SPLINE
SPL {X  -159.063, Y  +688.696, Z    +0.000, E1   -17.094, E3 +464723.597}
SPL {X  -159.987, Y  +672.488, Z    +0.000, E1    -5.638, E3 +464747.662}
SPL {X  -159.990, Y  +663.928, Z    +0.000, E1    +0.338, E3 +464753.456}
SPL {X  -159.990, Y  +658.009, Z    +0.000, E1    +4.774, E3 +464757.156}
SPL {X  -159.990, Y  +651.567, Z    +0.000, E1    +9.674, E3 +464762.560}
SPL {X  -159.990, Y  +638.711, Z    +0.000, E1   +17.883, E3 +464778.205}
SPL {X  -159.990, Y  +631.642, Z    +0.000, E1   +20.884, E3 +464793.764}
SPL {X  -159.990, Y  +626.048, Z    +0.000, E1   +22.026, E3 +464813.757}
SPL {X  -159.990, Y  +623.760, Z    +0.000, E1   +22.031, E3 +464825.745}
SPL {X  -159.990, Y  +621.334, Z    +0.000, E1   +22.029, E3 +464838.471}
SPL {X  -159.990, Y  +618.387, Z    +0.000, E1   +22.057, E3 +464853.861}
SPL {X  -159.990, Y  +615.830, Z    +0.000, E1   +22.023, E3 +464867.352}
SPL {X  -159.990, Y  +613.034, Z    +0.000, E1   +22.053, E3 +464881.959}
SPL {X  -159.990, Y  +609.503, Z    +0.000, E1   +22.054, E3 +464900.486}
SPL {X  -159.990, Y  +606.481, Z    +0.000, E1   +22.033, E3 +464916.360}
SPL {X  -159.990, Y  +603.419, Z    +0.000, E1   +22.064, E3 +464932.299}
SPL {X  -159.990, Y  +600.642, Z    +0.000, E1   +22.032, E3 +464946.929}
SPL {X  -159.990, Y  +598.568, Z    +0.000, E1   +22.046, E3 +464957.722}
SPL {X  -159.990, Y  +595.493, Z    +0.000, E1   +22.070, E3 +464973.805}
SPL {X  -159.990, Y  +592.865, Z    +0.000, E1   +22.036, E3 +464987.633}
SPL {X  -159.990, Y  +590.803, Z    +0.000, E1   +22.046, E3 +464998.424}
SPL {X  -159.990, Y  +587.778, Z    +0.000, E1   +22.073, E3 +465014.199}
SPL {X  -159.990, Y  +585.120, Z    +0.000, E1   +22.045, E3 +465028.143}
SPL {X  -159.990, Y  +583.118, Z    +0.000, E1   +22.052, E3 +465038.630}
SPL {X  -159.990, Y  +580.131, Z    +0.000, E1   +22.078, E3 +465054.236}
SPL {X  -159.990, Y  +576.888, Z    +0.000, E1   +22.061, E3 +465071.266}
SPL {X  -159.990, Y  +574.280, Z    +0.000, E1   +22.051, E3 +465084.940}
SPL {X  -159.990, Y  +572.375, Z    +0.000, E1   +22.037, E3 +465094.978}
SPL {X  -159.990, Y  +569.881, Z    +0.000, E1   +22.067, E3 +465107.973}
SPL {X  -159.990, Y  +567.211, Z    +0.000, E1   +22.046, E3 +465122.000}
SPL {X  -159.990, Y  +565.039, Z    +0.000, E1   +22.047, E3 +465133.377}
SPL {X  -159.990, Y  +562.755, Z    +0.000, E1   +22.047, E3 +465145.363}
SPL {X  -159.990, Y  +560.652, Z    +0.000, E1   +22.038, E3 +465156.408}
SPL {X  -159.990, Y  +558.852, Z    +0.000, E1   +22.046, E3 +465165.779}
SPL {X  -159.990, Y  +556.672, Z    +0.000, E1   +22.055, E3 +465177.169}
SPL {X  -159.990, Y  +553.726, Z    +0.000, E1   +22.080, E3 +465192.531}
SPL {X  -159.990, Y  +550.886, Z    +0.000, E1   +22.056, E3 +465207.470}
SPL {X  -159.990, Y  +548.814, Z    +0.000, E1   +22.049, E3 +465218.316}
SPL {X  -159.990, Y  +546.122, Z    +0.000, E1   +22.088, E3 +465232.330}
SPL {X  -159.990, Y  +542.390, Z    +0.000, E1   +22.086, E3 +465251.912}
SPL {X  -159.990, Y  +539.341, Z    +0.000, E1   +22.056, E3 +465267.933}
SPL {X  -159.990, Y  +536.984, Z    +0.000, E1   +22.057, E3 +465280.264}
SPL {X  -159.990, Y  +534.045, Z    +0.000, E1   +22.087, E3 +465295.589}
SPL {X  -159.990, Y  +530.476, Z    +0.000, E1   +22.084, E3 +465314.282}
SPL {X  -159.990, Y  +527.412, Z    +0.000, E1   +22.067, E3 +465330.346}
SPL {X  -159.990, Y  +525.349, Z    +0.000, E1   +22.050, E3 +465341.187}
SPL {X  -159.990, Y  +523.717, Z    +0.000, E1   +22.050, E3 +465349.752}
SPL {X  -159.990, Y  +521.599, Z    +0.000, E1   +22.060, E3 +465360.820}
SPL {X  -159.990, Y  +519.209, Z    +0.000, E1   +22.063, E3 +465373.295}
SPL {X  -159.990, Y  +517.330, Z    +0.000, E1   +22.053, E3 +465383.151}
SPL {X  -159.990, Y  +514.729, Z    +0.000, E1   +22.089, E3 +465396.709}
SPL {X  -159.990, Y  +511.670, Z    +0.000, E1   +22.064, E3 +465412.796}
SPL {X  -159.990, Y  +506.947, Z    +0.000, E1   +23.726, E3 +465422.825}
SPL {X  -159.990, Y  +496.921, Z    +0.000, E1   +28.340, E3 +465431.573}
SPL {X  -159.990, Y  +495.822, Z    +0.000, E1   +27.449, E3 +465442.321}
SPL {X  -159.990, Y  +494.952, Z    +0.000, E1   +26.628, E3 +465451.905}
SPL {X  -159.990, Y  +493.896, Z    +0.000, E1   +25.736, E3 +465463.234}
SPL {X  -159.990, Y  +491.647, Z    +0.000, E1   +25.401, E3 +465475.770}
SPL {X  -159.990, Y  +488.807, Z    +0.000, E1   +25.397, E3 +465488.468}
SPL {X  -159.990, Y  +486.070, Z    +0.000, E1   +25.399, E3 +465500.699}
SPL {X  -159.990, Y  +482.821, Z    +0.000, E1   +25.411, E3 +465515.201}
SPL {X  -159.990, Y  +480.183, Z    +0.000, E1   +25.384, E3 +465527.041}
SPL {X  -159.990, Y  +477.508, Z    +0.000, E1   +25.410, E3 +465538.950}
SPL {X  -159.990, Y  +473.634, Z    +0.000, E1   +25.426, E3 +465556.239}
SPL {X  -159.990, Y  +470.047, Z    +0.000, E1   +25.402, E3 +465572.320}
SPL {X  -159.990, Y  +467.082, Z    +0.000, E1   +25.399, E3 +465585.567}
SPL {X  -159.990, Y  +464.063, Z    +0.000, E1   +25.405, E3 +465599.062}
SPL {X  -159.990, Y  +460.712, Z    +0.000, E1   +25.411, E3 +465614.022}
SPL {X  -159.990, Y  +457.497, Z    +0.000, E1   +25.403, E3 +465628.394}
SPL {X  -159.990, Y  +455.126, Z    +0.000, E1   +25.389, E3 +465639.002}
SPL {X  -159.990, Y  +453.438, Z    +0.000, E1   +25.385, E3 +465646.562}
SPL {X  -159.990, Y  +450.823, Z    +0.000, E1   +25.417, E3 +465658.182}
SPL {X  -159.990, Y  +446.894, Z    +0.000, E1   +25.428, E3 +465675.739}
SPL {X  -159.990, Y  +443.345, Z    +0.000, E1   +25.390, E3 +465691.746}
SPL {X  -159.990, Y  +441.077, Z    +0.000, E1   +25.369, E3 +465701.945}
SPL {X  -159.990, Y  +438.608, Z    +0.000, E1   +25.392, E3 +465712.941}
SPL {X  -159.990, Y  +434.852, Z    +0.000, E1   +25.415, E3 +465729.696}
SPL {X  -159.990, Y  +430.645, Z    +0.000, E1   +25.414, E3 +465748.515}
SPL {X  -159.990, Y  +426.865, Z    +0.000, E1   +25.398, E3 +465765.445}
SPL {X  -159.990, Y  +424.251, Z    +0.000, E1   +25.375, E3 +465777.182}
SPL {X  -159.990, Y  +421.010, Z    +0.000, E1   +25.418, E3 +465791.597}
SPL {X  -159.990, Y  +417.514, Z    +0.000, E1   +25.386, E3 +465807.290}
SPL {X  -159.990, Y  +414.805, Z    +0.000, E1   +25.385, E3 +465819.410}
SPL {X  -159.990, Y  +411.959, Z    +0.000, E1   +25.386, E3 +465832.137}
SPL {X  -159.990, Y  +408.981, Z    +0.000, E1   +25.392, E3 +465845.440}
SPL {X  -159.990, Y  +406.574, Z    +0.000, E1   +25.375, E3 +465856.214}
SPL {X  -159.990, Y  +403.513, Z    +0.000, E1   +25.420, E3 +465869.813}
SPL {X  -159.990, Y  +399.257, Z    +0.000, E1   +25.420, E3 +465888.854}
SPL {X  -159.990, Y  +395.992, Z    +0.000, E1   +25.380, E3 +465903.544}
SPL {X  -159.990, Y  +393.569, Z    +0.000, E1   +25.379, E3 +465914.387}
SPL {X  -159.990, Y  +390.564, Z    +0.000, E1   +25.393, E3 +465927.831}
SPL {X  -159.990, Y  +387.503, Z    +0.000, E1   +25.378, E3 +465941.546}
SPL {X  -159.990, Y  +384.900, Z    +0.000, E1   +25.383, E3 +465953.156}
SPL {X  -159.990, Y  +382.110, Z    +0.000, E1   +25.393, E3 +465965.602}
SPL {X  -159.961, Y  +379.439, Z    +0.000, E1   +25.380, E3 +465977.582}
SPL {X  -159.894, Y  +376.959, Z    +0.000, E1   +25.370, E3 +465988.759}
SPL {X  -159.784, Y  +374.382, Z    +0.000, E1   +25.356, E3 +466000.399}
SPL {X  -159.621, Y  +371.640, Z    +0.000, E1   +25.335, E3 +466012.839}
SPL {X  -159.406, Y  +368.844, Z    +0.000, E1   +25.307, E3 +466025.552}
SPL {X  -159.144, Y  +366.072, Z    +0.000, E1   +25.281, E3 +466038.160}
SPL {X  -158.822, Y  +363.200, Z    +0.000, E1   +25.236, E3 +466051.333}
SPL {X  -158.491, Y  +360.654, Z    +0.000, E1   +25.188, E3 +466063.073}
SPL {X  -158.127, Y  +358.155, Z    +0.000, E1   +25.126, E3 +466074.692}
SPL {X  -158.095, Y  +357.947, Z    +0.000, E1   +21.741, E3 +466106.265}
ENDSPLINE

SPLINE
SPL {X  -158.454, Y  +360.384, Z    +0.000, E1   +19.366, E3 +466118.416}
SPL {X  -159.737, Y  +373.507, Z    +0.000, E1   +10.311, E3 +466140.451}
SPL {X  -159.990, Y  +382.574, Z    +0.000, E1    +4.463, E3 +466147.139}
SPL {X  -159.990, Y  +387.496, Z    +0.000, E1    +1.004, E3 +466149.884}
SPL {X  -159.990, Y  +395.121, Z    +0.000, E1    -4.514, E3 +466154.196}
SPL {X  -159.990, Y  +407.941, Z    +0.000, E1   -14.126, E3 +466166.270}
SPL {X  -159.990, Y  +418.671, Z    +0.000, E1   -19.855, E3 +466185.687}
SPL {X  -159.990, Y  +429.878, Z    +0.000, E1   -23.330, E3 +466215.742}
SPL {X  -159.990, Y  +432.766, Z    +0.000, E1   -23.321, E3 +466229.964}
SPL {X  -159.990, Y  +434.794, Z    +0.000, E1   -23.304, E3 +466239.996}
SPL {X  -159.990, Y  +437.007, Z    +0.000, E1   -23.323, E3 +466250.848}
SPL {X  -159.990, Y  +439.778, Z    +0.000, E1   -23.323, E3 +466264.480}
SPL {X  -159.990, Y  +442.010, Z    +0.000, E1   -23.308, E3 +466275.501}
SPL {X  -159.990, Y  +443.729, Z    +0.000, E1   -23.310, E3 +466283.958}
SPL {X  -159.990, Y  +446.037, Z    +0.000, E1   -23.324, E3 +466295.295}
SPL {X  -159.990, Y  +449.434, Z    +0.000, E1   -23.356, E3 +466311.916}
SPL {X  -159.990, Y  +453.256, Z    +0.000, E1   -23.349, E3 +466330.751}
SPL {X  -159.990, Y  +455.953, Z    +0.000, E1   -23.320, E3 +466344.065}
SPL {X  -159.990, Y  +458.265, Z    +0.000, E1   -23.328, E3 +466355.420}
SPL {X  -159.990, Y  +460.492, Z    +0.000, E1   -23.317, E3 +466366.419}
SPL {X  -159.990, Y  +462.929, Z    +0.000, E1   -23.331, E3 +466378.375}
SPL {X  -159.990, Y  +466.197, Z    +0.000, E1   -23.351, E3 +466394.412}
SPL {X  -159.990, Y  +468.951, Z    +0.000, E1   -23.319, E3 +466408.029}
SPL {X  -159.990, Y  +470.991, Z    +0.000, E1   -23.322, E3 +466418.059}
SPL {X  -159.990, Y  +474.027, Z    +0.000, E1   -23.352, E3 +466432.963}
SPL {X  -159.990, Y  +476.830, Z    +0.000, E1   -23.323, E3 +466446.830}
SPL {X  -159.990, Y  +479.553, Z    +0.000, E1   -23.328, E3 +466460.233}
SPL {X  -159.990, Y  +482.950, Z    +0.000, E1   -23.350, E3 +466476.905}
SPL {X  -159.990, Y  +486.109, Z    +0.000, E1   -23.322, E3 +466492.520}
SPL {X  -159.990, Y  +488.481, Z    +0.000, E1   -23.319, E3 +466504.200}
SPL {X  -159.990, Y  +491.454, Z    +0.000, E1   -23.343, E3 +466518.780}
SPL {X  -159.990, Y  +494.937, Z    +0.000, E1   -23.343, E3 +466535.924}
SPL {X  -159.990, Y  +497.668, Z    +0.000, E1   -23.317, E3 +466549.418}
SPL {X  -159.990, Y  +499.995, Z    +0.000, E1   -23.324, E3 +466560.855}
SPL {X  -159.990, Y  +502.456, Z    +0.000, E1   -23.324, E3 +466572.970}
SPL {X  -159.990, Y  +504.508, Z    +0.000, E1   -23.311, E3 +466583.104}
SPL {X  -159.990, Y  +506.420, Z    +0.000, E1   -23.317, E3 +466592.497}
SPL {X  -159.990, Y  +508.862, Z    +0.000, E1   -23.328, E3 +466604.490}
SPL {X  -159.990, Y  +511.771, Z    +0.000, E1   -23.331, E3 +466618.811}
SPL {X  -159.990, Y  +514.016, Z    +0.000, E1   -23.308, E3 +466629.915}
SPL {X  -159.990, Y  +516.860, Z    +0.000, E1   -23.355, E3 +466643.801}
SPL {X  -159.990, Y  +520.719, Z    +0.000, E1   -23.363, E3 +466662.712}
SPL {X  -159.990, Y  +523.968, Z    +0.000, E1   -23.332, E3 +466678.797}
SPL {X  -159.990, Y  +526.466, Z    +0.000, E1   -23.320, E3 +466691.140}
SPL {X  -159.990, Y  +528.815, Z    +0.000, E1   -23.322, E3 +466702.699}
SPL {X  -159.990, Y  +531.246, Z    +0.000, E1   -23.325, E3 +466714.638}
SPL {X  -159.990, Y  +534.143, Z    +0.000, E1   -23.341, E3 +466728.873}
SPL {X  -159.990, Y  +537.024, Z    +0.000, E1   -23.321, E3 +466743.116}
SPL {X  -159.990, Y  +539.129, Z    +0.000, E1   -23.310, E3 +466753.499}
SPL {X  -159.990, Y  +541.882, Z    +0.000, E1   -23.346, E3 +466766.980}
SPL {X  -159.990, Y  +544.941, Z    +0.000, E1   -23.325, E3 +466782.063}
SPL {X  -159.990, Y  +547.390, Z    +0.000, E1   -23.325, E3 +466794.116}
SPL {X  -159.990, Y  +550.708, Z    +0.000, E1   -23.357, E3 +466810.383}
SPL {X  -159.990, Y  +553.642, Z    +0.000, E1   -23.319, E3 +466824.890}
SPL {X  -159.990, Y  +555.637, Z    +0.000, E1   -23.323, E3 +466834.704}
SPL {X  -159.990, Y  +558.758, Z    +0.000, E1   -23.351, E3 +466850.014}
SPL {X  -159.990, Y  +561.830, Z    +0.000, E1   -23.325, E3 +466865.187}
SPL {X  -159.990, Y  +564.273, Z    +0.000, E1   -23.325, E3 +466877.212}
SPL {X  -159.990, Y  +567.351, Z    +0.000, E1   -23.348, E3 +466892.307}
SPL {X  -159.990, Y  +570.560, Z    +0.000, E1   -23.333, E3 +466908.137}
SPL {X  -159.990, Y  +572.975, Z    +0.000, E1   -23.316, E3 +466920.056}
SPL {X  -159.990, Y  +575.097, Z    +0.000, E1   -23.325, E3 +466930.483}
SPL {X  -159.990, Y  +578.356, Z    +0.000, E1   -23.358, E3 +466946.455}
SPL {X  -159.990, Y  +582.292, Z    +0.000, E1   -23.360, E3 +466965.771}
SPL {X  -159.990, Y  +585.165, Z    +0.000, E1   -23.322, E3 +466980.014}
SPL {X  -159.990, Y  +587.388, Z    +0.000, E1   -23.328, E3 +466990.927}
SPL {X  -159.990, Y  +589.763, Z    +0.000, E1   -23.328, E3 +467002.614}
SPL {X  -159.990, Y  +592.397, Z    +0.000, E1   -23.344, E3 +467015.495}
SPL {X  -159.990, Y  +595.589, Z    +0.000, E1   -23.356, E3 +467031.167}
SPL {X  -159.990, Y  +598.571, Z    +0.000, E1   -23.347, E3 +467045.811}
SPL {X  -159.990, Y  +600.935, Z    +0.000, E1   -23.343, E3 +467057.404}
SPL {X  -159.990, Y  +603.047, Z    +0.000, E1   -23.344, E3 +467067.790}
SPL {X  -159.990, Y  +605.187, Z    +0.000, E1   -23.344, E3 +467078.311}
SPL {X  -159.990, Y  +607.319, Z    +0.000, E1   -23.353, E3 +467088.774}
SPL {X  -159.990, Y  +609.514, Z    +0.000, E1   -23.337, E3 +467099.603}
SPL {X  -159.990, Y  +611.376, Z    +0.000, E1   -23.336, E3 +467108.790}
SPL {X  -159.990, Y  +613.591, Z    +0.000, E1   -23.342, E3 +467119.667}
SPL {X  -159.990, Y  +615.604, Z    +0.000, E1   -23.330, E3 +467129.605}
SPL {X  -159.990, Y  +617.623, Z    +0.000, E1   -23.337, E3 +467139.535}
SPL {X  -159.990, Y  +620.788, Z    +0.000, E1   -23.368, E3 +467155.041}
SPL {X  -159.990, Y  +623.764, Z    +0.000, E1   -23.335, E3 +467169.733}
SPL {X  -159.990, Y  +625.941, Z    +0.000, E1   -23.337, E3 +467180.424}
SPL {X  -159.990, Y  +628.611, Z    +0.000, E1   -23.357, E3 +467193.503}
SPL {X  -159.990, Y  +631.169, Z    +0.000, E1   -23.338, E3 +467206.107}
SPL {X  -159.990, Y  +633.318, Z    +0.000, E1   -23.339, E3 +467216.697}
SPL {X  -159.990, Y  +635.650, Z    +0.000, E1   -23.339, E3 +467228.167}
SPL {X  -159.990, Y  +637.839, Z    +0.000, E1   -23.335, E3 +467238.978}
SPL {X  -159.990, Y  +640.072, Z    +0.000, E1   -23.325, E3 +467250.010}
SPL {X  -159.990, Y  +642.230, Z    +0.000, E1   -23.323, E3 +467260.691}
SPL {X  -159.990, Y  +645.287, Z    +0.000, E1   -23.340, E3 +467275.717}
SPL {X  -159.990, Y  +647.803, Z    +0.000, E1   -23.310, E3 +467288.194}
SPL {X  -159.990, Y  +650.790, Z    +0.000, E1   -23.346, E3 +467302.802}
SPL {X  -159.990, Y  +654.543, Z    +0.000, E1   -23.348, E3 +467321.255}
SPL {X  -159.990, Y  +658.319, Z    +0.000, E1   -23.349, E3 +467339.844}
SPL {X  -159.990, Y  +661.392, Z    +0.000, E1   -23.318, E3 +467355.047}
SPL {X  -159.990, Y  +663.662, Z    +0.000, E1   -23.322, E3 +467366.172}
SPL {X  -159.990, Y  +665.964, Z    +0.000, E1   -23.328, E3 +467377.462}
SPL {X  -159.990, Y  +667.870, Z    +0.000, E1   -23.320, E3 +467386.869}
SPL {X  -159.990, Y  +669.861, Z    +0.000, E1   -23.321, E3 +467396.670}
SPL {X  -159.990, Y  +671.893, Z    +0.000, E1   -23.319, E3 +467406.678}
SPL {X  -159.974, Y  +673.789, Z    +0.000, E1   -23.323, E3 +467415.994}
SPL {X  -159.924, Y  +676.110, Z    +0.000, E1   -23.320, E3 +467427.478}
SPL {X  -159.801, Y  +679.265, Z    +0.000, E1   -23.327, E3 +467443.097}
SPL {X  -159.626, Y  +682.287, Z    +0.000, E1   -23.280, E3 +467458.195}
SPL {X  -159.462, Y  +684.486, Z    +0.000, E1   -23.258, E3 +467469.195}
SPL {X  -159.246, Y  +686.911, Z    +0.000, E1   -23.230, E3 +467481.356}
SPL {X  -159.019, Y  +689.098, Z    +0.000, E1   -23.200, E3 +467492.358}
SPL {X  -158.660, Y  +692.086, Z    +0.000, E1   -23.176, E3 +467507.402}
ENDSPLINE

SPLINE
SPL {X  -159.063, Y  +688.696, Z    +0.000, E1   -17.094, E3 +467549.684}
SPL {X  -159.967, Y  +674.206, Z    +0.000, E1    -6.731, E3 +467572.496}
SPL {X  -159.990, Y  +665.270, Z    +0.000, E1    -0.699, E3 +467578.666}
SPL {X  -159.990, Y  +658.009, Z    +0.000, E1    +4.774, E3 +467583.243}
SPL {X  -159.990, Y  +651.567, Z    +0.000, E1    +9.674, E3 +467588.647}
SPL {X  -159.990, Y  +638.711, Z    +0.000, E1   +17.883, E3 +467604.292}
SPL {X  -159.990, Y  +631.642, Z    +0.000, E1   +20.884, E3 +467619.851}
SPL {X  -159.990, Y  +626.048, Z    +0.000, E1   +22.026, E3 +467639.844}
SPL {X  -159.990, Y  +623.760, Z    +0.000, E1   +22.031, E3 +467651.832}
SPL {X  -159.990, Y  +621.334, Z    +0.000, E1   +22.029, E3 +467664.558}
SPL {X  -159.990, Y  +618.387, Z    +0.000, E1   +22.057, E3 +467679.948}
SPL {X  -159.990, Y  +614.928, Z    +0.000, E1   +22.055, E3 +467698.101}
SPL {X  -159.990, Y  +611.459, Z    +0.000, E1   +22.053, E3 +467716.304}
SPL {X  -159.990, Y  +608.810, Z    +0.000, E1   +22.023, E3 +467730.271}
SPL {X  -159.990, Y  +606.481, Z    +0.000, E1   +22.033, E3 +467742.447}
SPL {X  -159.990, Y  +603.419, Z    +0.000, E1   +22.064, E3 +467758.386}
SPL {X  -159.990, Y  +600.642, Z    +0.000, E1   +22.032, E3 +467773.016}
SPL {X  -159.990, Y  +598.568, Z    +0.000, E1   +22.046, E3 +467783.809}
SPL {X  -159.990, Y  +596.440, Z    +0.000, E1   +22.036, E3 +467794.990}
SPL {X  -159.990, Y  +593.768, Z    +0.000, E1   +22.071, E3 +467808.923}
SPL {X  -159.990, Y  +590.803, Z    +0.000, E1   +22.046, E3 +467824.511}
SPL {X  -159.990, Y  +587.778, Z    +0.000, E1   +22.073, E3 +467840.286}
SPL {X  -159.990, Y  +585.120, Z    +0.000, E1   +22.045, E3 +467854.230}
SPL {X  -159.990, Y  +583.118, Z    +0.000, E1   +22.052, E3 +467864.717}
SPL {X  -159.990, Y  +580.131, Z    +0.000, E1   +22.078, E3 +467880.323}
SPL {X  -159.990, Y  +576.888, Z    +0.000, E1   +22.061, E3 +467897.353}
SPL {X  -159.990, Y  +574.280, Z    +0.000, E1   +22.051, E3 +467911.027}
SPL {X  -159.990, Y  +572.375, Z    +0.000, E1   +22.037, E3 +467921.065}
SPL {X  -159.990, Y  +569.881, Z    +0.000, E1   +22.067, E3 +467934.059}
SPL {X  -159.990, Y  +567.211, Z    +0.000, E1   +22.046, E3 +467948.087}
SPL {X  -159.990, Y  +565.039, Z    +0.000, E1   +22.047, E3 +467959.464}
SPL {X  -159.990, Y  +562.755, Z    +0.000, E1   +22.047, E3 +467971.449}
SPL {X  -159.990, Y  +559.661, Z    +0.000, E1   +22.078, E3 +467987.581}
SPL {X  -159.990, Y  +555.965, Z    +0.000, E1   +22.085, E3 +468006.890}
SPL {X  -159.990, Y  +553.115, Z    +0.000, E1   +22.054, E3 +468021.876}
SPL {X  -159.990, Y  +550.886, Z    +0.000, E1   +22.056, E3 +468033.557}
SPL {X  -159.990, Y  +547.986, Z    +0.000, E1   +22.078, E3 +468048.677}
SPL {X  -159.990, Y  +545.350, Z    +0.000, E1   +22.053, E3 +468062.538}
SPL {X  -159.990, Y  +543.405, Z    +0.000, E1   +22.048, E3 +468072.751}
SPL {X  -159.990, Y  +541.673, Z    +0.000, E1   +22.053, E3 +468081.815}
SPL {X  -159.990, Y  +539.341, Z    +0.000, E1   +22.056, E3 +468094.020}
SPL {X  -159.990, Y  +536.301, Z    +0.000, E1   +22.084, E3 +468109.875}
SPL {X  -159.990, Y  +533.389, Z    +0.000, E1   +22.057, E3 +468125.182}
SPL {X  -159.990, Y  +531.347, Z    +0.000, E1   +22.052, E3 +468135.883}
SPL {X  -159.990, Y  +529.626, Z    +0.000, E1   +22.051, E3 +468144.880}
SPL {X  -159.990, Y  +527.412, Z    +0.000, E1   +22.067, E3 +468156.432}
SPL {X  -159.990, Y  +524.425, Z    +0.000, E1   +22.078, E3 +468172.065}
SPL {X  -159.990, Y  +521.599, Z    +0.000, E1   +22.060, E3 +468186.907}
SPL {X  -159.990, Y  +519.209, Z    +0.000, E1   +22.063, E3 +468199.382}
SPL {X  -159.990, Y  +516.651, Z    +0.000, E1   +22.071, E3 +468212.761}
SPL {X  -159.990, Y  +514.122, Z    +0.000, E1   +22.061, E3 +468226.033}
SPL {X  -159.990, Y  +511.670, Z    +0.000, E1   +22.064, E3 +468238.883}
SPL {X  -159.990, Y  +506.947, Z    +0.000, E1   +23.726, E3 +468248.912}
SPL {X  -159.990, Y  +496.921, Z    +0.000, E1   +28.340, E3 +468257.660}
SPL {X  -159.990, Y  +495.822, Z    +0.000, E1   +27.449, E3 +468268.408}
SPL {X  -159.990, Y  +494.952, Z    +0.000, E1   +26.628, E3 +468277.992}
SPL {X  -159.990, Y  +493.896, Z    +0.000, E1   +25.736, E3 +468289.321}
SPL {X  -159.990, Y  +491.647, Z    +0.000, E1   +25.401, E3 +468301.857}
SPL {X  -159.990, Y  +488.807, Z    +0.000, E1   +25.397, E3 +468314.555}
SPL {X  -159.990, Y  +486.070, Z    +0.000, E1   +25.399, E3 +468326.786}
SPL {X  -159.990, Y  +483.747, Z    +0.000, E1   +25.384, E3 +468337.199}
SPL {X  -159.990, Y  +481.980, Z    +0.000, E1   +25.384, E3 +468345.097}
SPL {X  -159.990, Y  +479.252, Z    +0.000, E1   +25.412, E3 +468357.238}
SPL {X  -159.990, Y  +475.940, Z    +0.000, E1   +25.403, E3 +468372.059}
SPL {X  -159.990, Y  +473.026, Z    +0.000, E1   +25.399, E3 +468385.088}
SPL {X  -159.990, Y  +470.047, Z    +0.000, E1   +25.402, E3 +468398.407}
SPL {X  -159.990, Y  +466.213, Z    +0.000, E1   +25.433, E3 +468415.486}
SPL {X  -159.990, Y  +462.520, Z    +0.000, E1   +25.400, E3 +468432.055}
SPL {X  -159.990, Y  +460.081, Z    +0.000, E1   +25.390, E3 +468442.956}
SPL {X  -159.990, Y  +457.497, Z    +0.000, E1   +25.403, E3 +468454.481}
SPL {X  -159.990, Y  +455.126, Z    +0.000, E1   +25.389, E3 +468465.089}
SPL {X  -159.990, Y  +452.123, Z    +0.000, E1   +25.426, E3 +468478.447}
SPL {X  -159.990, Y  +448.503, Z    +0.000, E1   +25.410, E3 +468494.648}
SPL {X  -159.990, Y  +445.882, Z    +0.000, E1   +25.385, E3 +468506.451}
SPL {X  -159.990, Y  +443.345, Z    +0.000, E1   +25.390, E3 +468517.833}
SPL {X  -159.990, Y  +441.077, Z    +0.000, E1   +25.369, E3 +468528.032}
SPL {X  -159.990, Y  +438.608, Z    +0.000, E1   +25.392, E3 +468539.028}
SPL {X  -159.990, Y  +434.852, Z    +0.000, E1   +25.415, E3 +468555.783}
SPL {X  -159.990, Y  +430.645, Z    +0.000, E1   +25.414, E3 +468574.602}
SPL {X  -159.990, Y  +426.865, Z    +0.000, E1   +25.398, E3 +468591.532}
SPL {X  -159.990, Y  +424.251, Z    +0.000, E1   +25.375, E3 +468603.269}
SPL {X  -159.990, Y  +421.010, Z    +0.000, E1   +25.418, E3 +468617.684}
SPL {X  -159.990, Y  +417.514, Z    +0.000, E1   +25.386, E3 +468633.377}
SPL {X  -159.990, Y  +414.805, Z    +0.000, E1   +25.385, E3 +468645.497}
SPL {X  -159.990, Y  +411.282, Z    +0.000, E1   +25.413, E3 +468661.198}
SPL {X  -159.990, Y  +408.351, Z    +0.000, E1   +25.372, E3 +468674.385}
SPL {X  -159.990, Y  +405.773, Z    +0.000, E1   +25.398, E3 +468685.837}
SPL {X  -159.990, Y  +402.805, Z    +0.000, E1   +25.389, E3 +468699.123}
SPL {X  -159.990, Y  +400.083, Z    +0.000, E1   +25.388, E3 +468711.300}
SPL {X  -159.990, Y  +396.740, Z    +0.000, E1   +25.410, E3 +468726.224}
SPL {X  -159.990, Y  +392.622, Z    +0.000, E1   +25.413, E3 +468744.652}
SPL {X  -159.990, Y  +388.328, Z    +0.000, E1   +25.413, E3 +468763.881}
SPL {X  -159.990, Y  +384.900, Z    +0.000, E1   +25.383, E3 +468779.243}
SPL {X  -159.990, Y  +382.110, Z    +0.000, E1   +25.393, E3 +468791.689}
SPL {X  -159.961, Y  +379.439, Z    +0.000, E1   +25.380, E3 +468803.669}
SPL {X  -159.894, Y  +376.959, Z    +0.000, E1   +25.370, E3 +468814.846}
SPL {X  -159.784, Y  +374.382, Z    +0.000, E1   +25.356, E3 +468826.486}
SPL {X  -159.621, Y  +371.640, Z    +0.000, E1   +25.335, E3 +468838.926}
SPL {X  -159.406, Y  +368.844, Z    +0.000, E1   +25.307, E3 +468851.639}
SPL {X  -159.144, Y  +366.072, Z    +0.000, E1   +25.281, E3 +468864.247}
SPL {X  -158.822, Y  +363.200, Z    +0.000, E1   +25.236, E3 +468877.420}
SPL {X  -158.491, Y  +360.654, Z    +0.000, E1   +25.188, E3 +468889.160}
SPL {X  -158.127, Y  +358.155, Z    +0.000, E1   +25.126, E3 +468900.779}
SPL {X  -158.095, Y  +357.947, Z    +0.000, E1   +21.741, E3 +468932.352}
ENDSPLINE

SPLINE
SPL {X  -158.454, Y  +360.384, Z    +0.000, E1   +19.366, E3 +468944.503}
SPL {X  -159.737, Y  +373.507, Z    +0.000, E1   +10.311, E3 +468966.538}
SPL {X  -159.990, Y  +382.574, Z    +0.000, E1    +4.463, E3 +468973.226}
SPL {X  -159.990, Y  +389.909, Z    +0.000, E1    -0.662, E3 +468977.240}
SPL {X  -159.990, Y  +396.289, Z    +0.000, E1    -5.500, E3 +468981.020}
SPL {X  -159.990, Y  +407.941, Z    +0.000, E1   -14.126, E3 +468992.357}
SPL {X  -159.990, Y  +418.671, Z    +0.000, E1   -19.855, E3 +469011.774}
SPL {X  -159.990, Y  +429.878, Z    +0.000, E1   -23.330, E3 +469041.829}
SPL {X  -159.990, Y  +432.103, Z    +0.000, E1   -23.301, E3 +469052.847}
SPL {X  -159.990, Y  +434.188, Z    +0.000, E1   -23.325, E3 +469063.044}
SPL {X  -159.990, Y  +437.007, Z    +0.000, E1   -23.323, E3 +469076.935}
SPL {X  -159.990, Y  +439.778, Z    +0.000, E1   -23.323, E3 +469090.567}
SPL {X  -159.990, Y  +442.945, Z    +0.000, E1   -23.339, E3 +469106.131}
SPL {X  -159.990, Y  +446.037, Z    +0.000, E1   -23.324, E3 +469121.382}
SPL {X  -159.990, Y  +448.797, Z    +0.000, E1   -23.331, E3 +469134.912}
SPL {X  -159.990, Y  +451.747, Z    +0.000, E1   -23.333, E3 +469149.460}
SPL {X  -159.990, Y  +454.210, Z    +0.000, E1   -23.316, E3 +469161.591}
SPL {X  -159.990, Y  +455.953, Z    +0.000, E1   -23.320, E3 +469170.152}
SPL {X  -159.990, Y  +458.265, Z    +0.000, E1   -23.328, E3 +469181.507}
SPL {X  -159.990, Y  +461.258, Z    +0.000, E1   -23.344, E3 +469196.223}
SPL {X  -159.990, Y  +464.382, Z    +0.000, E1   -23.332, E3 +469211.604}
SPL {X  -159.990, Y  +466.881, Z    +0.000, E1   -23.322, E3 +469223.924}
SPL {X  -159.990, Y  +468.951, Z    +0.000, E1   -23.319, E3 +469234.116}
SPL {X  -159.990, Y  +470.991, Z    +0.000, E1   -23.322, E3 +469244.146}
SPL {X  -159.990, Y  +474.027, Z    +0.000, E1   -23.352, E3 +469259.050}
SPL {X  -159.990, Y  +477.600, Z    +0.000, E1   -23.351, E3 +469276.653}
SPL {X  -159.990, Y  +481.169, Z    +0.000, E1   -23.337, E3 +469294.250}
SPL {X  -159.990, Y  +483.782, Z    +0.000, E1   -23.316, E3 +469307.155}
SPL {X  -159.990, Y  +486.109, Z    +0.000, E1   -23.322, E3 +469318.607}
SPL {X  -159.990, Y  +489.247, Z    +0.000, E1   -23.348, E3 +469333.995}
SPL {X  -159.990, Y  +493.031, Z    +0.000, E1   -23.350, E3 +469352.619}
SPL {X  -159.990, Y  +496.869, Z    +0.000, E1   -23.349, E3 +469371.509}
SPL {X  -159.990, Y  +499.995, Z    +0.000, E1   -23.324, E3 +469386.942}
SPL {X  -159.990, Y  +502.456, Z    +0.000, E1   -23.324, E3 +469399.057}
SPL {X  -159.990, Y  +505.646, Z    +0.000, E1   -23.350, E3 +469414.712}
SPL {X  -159.990, Y  +508.862, Z    +0.000, E1   -23.328, E3 +469430.577}
SPL {X  -159.990, Y  +510.971, Z    +0.000, E1   -23.308, E3 +469441.004}
SPL {X  -159.990, Y  +512.484, Z    +0.000, E1   -23.309, E3 +469448.454}
SPL {X  -159.990, Y  +514.757, Z    +0.000, E1   -23.329, E3 +469459.606}
SPL {X  -159.990, Y  +517.536, Z    +0.000, E1   -23.326, E3 +469473.273}
SPL {X  -159.990, Y  +519.961, Z    +0.000, E1   -23.334, E3 +469485.125}
SPL {X  -159.990, Y  +521.849, Z    +0.000, E1   -23.320, E3 +469494.448}
SPL {X  -159.990, Y  +523.968, Z    +0.000, E1   -23.332, E3 +469504.883}
SPL {X  -159.990, Y  +526.466, Z    +0.000, E1   -23.320, E3 +469517.227}
SPL {X  -159.990, Y  +528.815, Z    +0.000, E1   -23.322, E3 +469528.786}
SPL {X  -159.990, Y  +531.246, Z    +0.000, E1   -23.325, E3 +469540.725}
SPL {X  -159.990, Y  +533.354, Z    +0.000, E1   -23.318, E3 +469551.110}
SPL {X  -159.990, Y  +534.931, Z    +0.000, E1   -23.312, E3 +469558.905}
SPL {X  -159.990, Y  +537.024, Z    +0.000, E1   -23.321, E3 +469569.203}
SPL {X  -159.990, Y  +539.129, Z    +0.000, E1   -23.310, E3 +469579.586}
SPL {X  -159.990, Y  +541.183, Z    +0.000, E1   -23.319, E3 +469589.683}
SPL {X  -159.990, Y  +544.314, Z    +0.000, E1   -23.352, E3 +469605.011}
SPL {X  -159.990, Y  +548.126, Z    +0.000, E1   -23.354, E3 +469623.767}
SPL {X  -159.990, Y  +551.344, Z    +0.000, E1   -23.327, E3 +469639.659}
SPL {X  -159.990, Y  +553.642, Z    +0.000, E1   -23.319, E3 +469650.977}
SPL {X  -159.990, Y  +556.481, Z    +0.000, E1   -23.354, E3 +469664.884}
SPL {X  -159.990, Y  +559.475, Z    +0.000, E1   -23.321, E3 +469679.690}
SPL {X  -159.990, Y  +561.830, Z    +0.000, E1   -23.325, E3 +469691.274}
SPL {X  -159.990, Y  +564.273, Z    +0.000, E1   -23.325, E3 +469703.299}
SPL {X  -159.990, Y  +566.342, Z    +0.000, E1   -23.314, E3 +469713.503}
SPL {X  -159.990, Y  +568.849, Z    +0.000, E1   -23.338, E3 +469725.798}
SPL {X  -159.990, Y  +572.204, Z    +0.000, E1   -23.344, E3 +469742.293}
SPL {X  -159.990, Y  +575.097, Z    +0.000, E1   -23.325, E3 +469756.570}
SPL {X  -159.990, Y  +577.540, Z    +0.000, E1   -23.325, E3 +469768.599}
SPL {X  -159.990, Y  +580.312, Z    +0.000, E1   -23.340, E3 +469782.180}
SPL {X  -159.990, Y  +583.018, Z    +0.000, E1   -23.331, E3 +469795.485}
SPL {X  -159.990, Y  +585.165, Z    +0.000, E1   -23.322, E3 +469806.101}
SPL {X  -159.990, Y  +587.388, Z    +0.000, E1   -23.328, E3 +469817.014}
SPL {X  -159.990, Y  +589.763, Z    +0.000, E1   -23.328, E3 +469828.701}
SPL {X  -159.990, Y  +592.397, Z    +0.000, E1   -23.344, E3 +469841.582}
SPL {X  -159.990, Y  +595.589, Z    +0.000, E1   -23.356, E3 +469857.254}
SPL {X  -159.990, Y  +598.571, Z    +0.000, E1   -23.347, E3 +469871.898}
SPL {X  -159.990, Y  +600.935, Z    +0.000, E1   -23.343, E3 +469883.491}
SPL {X  -159.990, Y  +603.047, Z    +0.000, E1   -23.344, E3 +469893.877}
SPL {X  -159.990, Y  +605.187, Z    +0.000, E1   -23.344, E3 +469904.398}
SPL {X  -159.990, Y  +607.319, Z    +0.000, E1   -23.353, E3 +469914.861}
SPL {X  -159.990, Y  +610.569, Z    +0.000, E1   -23.372, E3 +469930.826}
SPL {X  -159.990, Y  +613.591, Z    +0.000, E1   -23.342, E3 +469945.754}
SPL {X  -159.990, Y  +615.604, Z    +0.000, E1   -23.330, E3 +469955.692}
SPL {X  -159.990, Y  +618.445, Z    +0.000, E1   -23.368, E3 +469969.605}
SPL {X  -159.990, Y  +621.517, Z    +0.000, E1   -23.337, E3 +469984.770}
SPL {X  -159.990, Y  +623.764, Z    +0.000, E1   -23.335, E3 +469995.820}
SPL {X  -159.990, Y  +626.608, Z    +0.000, E1   -23.361, E3 +470009.745}
SPL {X  -159.990, Y  +630.271, Z    +0.000, E1   -23.375, E3 +470027.706}
SPL {X  -159.990, Y  +633.318, Z    +0.000, E1   -23.339, E3 +470042.784}
SPL {X  -159.990, Y  +635.650, Z    +0.000, E1   -23.339, E3 +470054.254}
SPL {X  -159.990, Y  +637.839, Z    +0.000, E1   -23.335, E3 +470065.065}
SPL {X  -159.990, Y  +640.072, Z    +0.000, E1   -23.325, E3 +470076.097}
SPL {X  -159.990, Y  +643.026, Z    +0.000, E1   -23.354, E3 +470090.637}
SPL {X  -159.990, Y  +646.970, Z    +0.000, E1   -23.346, E3 +470110.101}
SPL {X  -159.990, Y  +650.790, Z    +0.000, E1   -23.346, E3 +470128.889}
SPL {X  -159.990, Y  +654.543, Z    +0.000, E1   -23.348, E3 +470147.342}
SPL {X  -159.990, Y  +658.319, Z    +0.000, E1   -23.349, E3 +470165.931}
SPL {X  -159.990, Y  +661.392, Z    +0.000, E1   -23.318, E3 +470181.134}
SPL {X  -159.990, Y  +663.662, Z    +0.000, E1   -23.322, E3 +470192.258}
SPL {X  -159.990, Y  +665.964, Z    +0.000, E1   -23.328, E3 +470203.549}
SPL {X  -159.990, Y  +667.870, Z    +0.000, E1   -23.320, E3 +470212.956}
SPL {X  -159.990, Y  +669.861, Z    +0.000, E1   -23.321, E3 +470222.757}
SPL {X  -159.990, Y  +671.893, Z    +0.000, E1   -23.319, E3 +470232.765}
SPL {X  -159.974, Y  +673.789, Z    +0.000, E1   -23.323, E3 +470242.081}
SPL {X  -159.924, Y  +676.110, Z    +0.000, E1   -23.320, E3 +470253.565}
SPL {X  -159.801, Y  +679.265, Z    +0.000, E1   -23.327, E3 +470269.184}
SPL {X  -159.626, Y  +682.287, Z    +0.000, E1   -23.280, E3 +470284.282}
SPL {X  -159.462, Y  +684.486, Z    +0.000, E1   -23.258, E3 +470295.282}
SPL {X  -159.246, Y  +686.911, Z    +0.000, E1   -23.230, E3 +470307.443}
SPL {X  -159.019, Y  +689.098, Z    +0.000, E1   -23.200, E3 +470318.445}
SPL {X  -158.660, Y  +692.086, Z    +0.000, E1   -23.176, E3 +470333.489}
ENDSPLINE

SPLINE
SPL {X  -159.063, Y  +688.696, Z    +0.000, E1   -17.094, E3 +470375.771}
SPL {X  -159.967, Y  +674.206, Z    +0.000, E1    -6.731, E3 +470398.583}
SPL {X  -159.990, Y  +665.270, Z    +0.000, E1    -0.699, E3 +470404.753}
SPL {X  -159.990, Y  +658.009, Z    +0.000, E1    +4.774, E3 +470409.330}
SPL {X  -159.990, Y  +651.567, Z    +0.000, E1    +9.674, E3 +470414.734}
SPL {X  -159.990, Y  +637.762, Z    +0.000, E1   +18.345, E3 +470432.092}
SPL {X  -159.990, Y  +626.382, Z    +0.000, E1   +22.040, E3 +470464.141}
SPL {X  -159.990, Y  +623.760, Z    +0.000, E1   +22.031, E3 +470477.918}
SPL {X  -159.990, Y  +621.334, Z    +0.000, E1   +22.029, E3 +470490.645}
SPL {X  -159.990, Y  +618.387, Z    +0.000, E1   +22.057, E3 +470506.035}
SPL {X  -159.990, Y  +614.928, Z    +0.000, E1   +22.055, E3 +470524.187}
SPL {X  -159.990, Y  +611.459, Z    +0.000, E1   +22.053, E3 +470542.391}
SPL {X  -159.990, Y  +608.810, Z    +0.000, E1   +22.023, E3 +470556.358}
SPL {X  -159.990, Y  +606.481, Z    +0.000, E1   +22.033, E3 +470568.534}
SPL {X  -159.990, Y  +603.419, Z    +0.000, E1   +22.064, E3 +470584.473}
SPL {X  -159.990, Y  +600.642, Z    +0.000, E1   +22.032, E3 +470599.103}
SPL {X  -159.990, Y  +598.568, Z    +0.000, E1   +22.046, E3 +470609.896}
SPL {X  -159.990, Y  +595.493, Z    +0.000, E1   +22.070, E3 +470625.979}
SPL {X  -159.990, Y  +592.865, Z    +0.000, E1   +22.036, E3 +470639.807}
SPL {X  -159.990, Y  +590.803, Z    +0.000, E1   +22.046, E3 +470650.598}
SPL {X  -159.990, Y  +587.778, Z    +0.000, E1   +22.073, E3 +470666.373}
SPL {X  -159.990, Y  +585.120, Z    +0.000, E1   +22.045, E3 +470680.317}
SPL {X  -159.990, Y  +583.118, Z    +0.000, E1   +22.052, E3 +470690.804}
SPL {X  -159.990, Y  +580.131, Z    +0.000, E1   +22.078, E3 +470706.410}
SPL {X  -159.990, Y  +576.888, Z    +0.000, E1   +22.061, E3 +470723.440}
SPL {X  -159.990, Y  +574.280, Z    +0.000, E1   +22.051, E3 +470737.114}
SPL {X  -159.990, Y  +571.711, Z    +0.000, E1   +22.058, E3 +470750.588}
SPL {X  -159.990, Y  +569.285, Z    +0.000, E1   +22.044, E3 +470763.313}
SPL {X  -159.990, Y  +567.211, Z    +0.000, E1   +22.046, E3 +470774.174}
SPL {X  -159.990, Y  +565.039, Z    +0.000, E1   +22.047, E3 +470785.551}
SPL {X  -159.990, Y  +562.755, Z    +0.000, E1   +22.047, E3 +470797.536}
SPL {X  -159.990, Y  +560.652, Z    +0.000, E1   +22.038, E3 +470808.582}
SPL {X  -159.990, Y  +558.852, Z    +0.000, E1   +22.046, E3 +470817.953}
SPL {X  -159.990, Y  +556.672, Z    +0.000, E1   +22.055, E3 +470829.343}
SPL {X  -159.990, Y  +553.726, Z    +0.000, E1   +22.080, E3 +470844.705}
SPL {X  -159.990, Y  +550.886, Z    +0.000, E1   +22.056, E3 +470859.644}
SPL {X  -159.990, Y  +548.814, Z    +0.000, E1   +22.049, E3 +470870.490}
SPL {X  -159.990, Y  +546.122, Z    +0.000, E1   +22.088, E3 +470884.503}
SPL {X  -159.990, Y  +542.390, Z    +0.000, E1   +22.086, E3 +470904.085}
SPL {X  -159.990, Y  +539.341, Z    +0.000, E1   +22.056, E3 +470920.107}
SPL {X  -159.990, Y  +536.984, Z    +0.000, E1   +22.057, E3 +470932.438}
SPL {X  -159.990, Y  +534.045, Z    +0.000, E1   +22.087, E3 +470947.763}
SPL {X  -159.990, Y  +530.476, Z    +0.000, E1   +22.084, E3 +470966.456}
SPL {X  -159.990, Y  +527.412, Z    +0.000, E1   +22.067, E3 +470982.519}
SPL {X  -159.990, Y  +524.425, Z    +0.000, E1   +22.078, E3 +470998.152}
SPL {X  -159.990, Y  +521.599, Z    +0.000, E1   +22.060, E3 +471012.994}
SPL {X  -159.990, Y  +519.209, Z    +0.000, E1   +22.063, E3 +471025.469}
SPL {X  -159.990, Y  +516.651, Z    +0.000, E1   +22.071, E3 +471038.848}
SPL {X  -159.990, Y  +514.122, Z    +0.000, E1   +22.061, E3 +471052.120}
SPL {X  -159.990, Y  +511.670, Z    +0.000, E1   +22.064, E3 +471064.970}
SPL {X  -159.990, Y  +506.947, Z    +0.000, E1   +23.726, E3 +471074.999}
SPL {X  -159.990, Y  +496.921, Z    +0.000, E1   +28.340, E3 +471083.747}
SPL {X  -159.990, Y  +495.822, Z    +0.000, E1   +27.449, E3 +471094.495}
SPL {X  -159.990, Y  +494.952, Z    +0.000, E1   +26.628, E3 +471104.078}
SPL {X  -159.990, Y  +493.896, Z    +0.000, E1   +25.736, E3 +471115.408}
SPL {X  -159.990, Y  +491.647, Z    +0.000, E1   +25.401, E3 +471127.944}
SPL {X  -159.990, Y  +488.807, Z    +0.000, E1   +25.397, E3 +471140.642}
SPL {X  -159.990, Y  +486.070, Z    +0.000, E1   +25.399, E3 +471152.873}
SPL {X  -159.990, Y  +483.747, Z    +0.000, E1   +25.384, E3 +471163.286}
SPL {X  -159.990, Y  +481.980, Z    +0.000, E1   +25.384, E3 +471171.184}
SPL {X  -159.990, Y  +479.252, Z    +0.000, E1   +25.412, E3 +471183.325}
SPL {X  -159.990, Y  +475.940, Z    +0.000, E1   +25.403, E3 +471198.145}
SPL {X  -159.990, Y  +473.026, Z    +0.000, E1   +25.399, E3 +471211.175}
SPL {X  -159.990, Y  +470.047, Z    +0.000, E1   +25.402, E3 +471224.494}
SPL {X  -159.990, Y  +466.213, Z    +0.000, E1   +25.433, E3 +471241.573}
SPL {X  -159.990, Y  +462.520, Z    +0.000, E1   +25.400, E3 +471258.142}
SPL {X  -159.990, Y  +460.081, Z    +0.000, E1   +25.390, E3 +471269.043}
SPL {X  -159.990, Y  +457.497, Z    +0.000, E1   +25.403, E3 +471280.568}
SPL {X  -159.990, Y  +455.126, Z    +0.000, E1   +25.389, E3 +471291.176}
SPL {X  -159.990, Y  +452.123, Z    +0.000, E1   +25.426, E3 +471304.534}
SPL {X  -159.990, Y  +448.503, Z    +0.000, E1   +25.410, E3 +471320.735}
SPL {X  -159.990, Y  +445.882, Z    +0.000, E1   +25.385, E3 +471332.538}
SPL {X  -159.990, Y  +443.345, Z    +0.000, E1   +25.390, E3 +471343.920}
SPL {X  -159.990, Y  +441.077, Z    +0.000, E1   +25.369, E3 +471354.118}
SPL {X  -159.990, Y  +438.608, Z    +0.000, E1   +25.392, E3 +471365.115}
SPL {X  -159.990, Y  +435.579, Z    +0.000, E1   +25.386, E3 +471378.669}
SPL {X  -159.990, Y  +432.613, Z    +0.000, E1   +25.390, E3 +471391.937}
SPL {X  -159.990, Y  +429.079, Z    +0.000, E1   +25.407, E3 +471407.707}
SPL {X  -159.990, Y  +426.149, Z    +0.000, E1   +25.374, E3 +471420.869}
SPL {X  -159.990, Y  +423.417, Z    +0.000, E1   +25.400, E3 +471433.035}
SPL {X  -159.990, Y  +420.283, Z    +0.000, E1   +25.386, E3 +471447.079}
SPL {X  -159.990, Y  +417.514, Z    +0.000, E1   +25.386, E3 +471459.464}
SPL {X  -159.990, Y  +414.805, Z    +0.000, E1   +25.385, E3 +471471.584}
SPL {X  -159.990, Y  +411.282, Z    +0.000, E1   +25.413, E3 +471487.284}
SPL {X  -159.990, Y  +408.351, Z    +0.000, E1   +25.372, E3 +471500.472}
SPL {X  -159.990, Y  +405.773, Z    +0.000, E1   +25.398, E3 +471511.924}
SPL {X  -159.990, Y  +402.805, Z    +0.000, E1   +25.389, E3 +471525.210}
SPL {X  -159.990, Y  +400.083, Z    +0.000, E1   +25.388, E3 +471537.387}
SPL {X  -159.990, Y  +396.740, Z    +0.000, E1   +25.410, E3 +471552.311}
SPL {X  -159.990, Y  +392.622, Z    +0.000, E1   +25.413, E3 +471570.739}
SPL {X  -159.990, Y  +388.328, Z    +0.000, E1   +25.413, E3 +471589.967}
SPL {X  -159.990, Y  +384.900, Z    +0.000, E1   +25.383, E3 +471605.330}
SPL {X  -159.990, Y  +382.110, Z    +0.000, E1   +25.393, E3 +471617.776}
SPL {X  -159.961, Y  +379.439, Z    +0.000, E1   +25.380, E3 +471629.756}
SPL {X  -159.894, Y  +376.959, Z    +0.000, E1   +25.370, E3 +471640.933}
SPL {X  -159.784, Y  +374.382, Z    +0.000, E1   +25.356, E3 +471652.573}
SPL {X  -159.621, Y  +371.640, Z    +0.000, E1   +25.335, E3 +471665.013}
SPL {X  -159.406, Y  +368.844, Z    +0.000, E1   +25.307, E3 +471677.726}
SPL {X  -159.144, Y  +366.072, Z    +0.000, E1   +25.281, E3 +471690.334}
SPL {X  -158.822, Y  +363.200, Z    +0.000, E1   +25.236, E3 +471703.507}
SPL {X  -158.491, Y  +360.654, Z    +0.000, E1   +25.188, E3 +471715.247}
SPL {X  -158.127, Y  +358.155, Z    +0.000, E1   +25.126, E3 +471726.866}
SPL {X  -158.095, Y  +357.947, Z    +0.000, E1   +21.741, E3 +471758.439}
ENDSPLINE

SPLINE
SPL {X  -158.454, Y  +360.384, Z    +0.000, E1   +19.366, E3 +471770.590}
SPL {X  -159.737, Y  +373.507, Z    +0.000, E1   +10.311, E3 +471792.625}
SPL {X  -159.990, Y  +382.574, Z    +0.000, E1    +4.463, E3 +471799.313}
SPL {X  -159.990, Y  +387.496, Z    +0.000, E1    +1.004, E3 +471802.058}
SPL {X  -159.990, Y  +395.121, Z    +0.000, E1    -4.514, E3 +471806.370}
SPL {X  -159.990, Y  +407.941, Z    +0.000, E1   -14.126, E3 +471818.444}
SPL {X  -159.990, Y  +418.671, Z    +0.000, E1   -19.855, E3 +471837.861}
SPL {X  -159.990, Y  +429.878, Z    +0.000, E1   -23.330, E3 +471867.916}
SPL {X  -159.990, Y  +432.766, Z    +0.000, E1   -23.321, E3 +471882.138}
SPL {X  -159.990, Y  +434.794, Z    +0.000, E1   -23.304, E3 +471892.170}
SPL {X  -159.990, Y  +437.007, Z    +0.000, E1   -23.323, E3 +471903.022}
SPL {X  -159.990, Y  +439.778, Z    +0.000, E1   -23.323, E3 +471916.654}
SPL {X  -159.990, Y  +442.010, Z    +0.000, E1   -23.308, E3 +471927.675}
SPL {X  -159.990, Y  +443.729, Z    +0.000, E1   -23.310, E3 +471936.132}
SPL {X  -159.990, Y  +446.037, Z    +0.000, E1   -23.324, E3 +471947.469}
SPL {X  -159.990, Y  +448.797, Z    +0.000, E1   -23.331, E3 +471960.999}
SPL {X  -159.990, Y  +451.747, Z    +0.000, E1   -23.333, E3 +471975.547}
SPL {X  -159.990, Y  +455.185, Z    +0.000, E1   -23.350, E3 +471992.407}
SPL {X  -159.990, Y  +458.265, Z    +0.000, E1   -23.328, E3 +472007.594}
SPL {X  -159.990, Y  +460.492, Z    +0.000, E1   -23.317, E3 +472018.593}
SPL {X  -159.990, Y  +462.929, Z    +0.000, E1   -23.331, E3 +472030.548}
SPL {X  -159.990, Y  +465.027, Z    +0.000, E1   -23.313, E3 +472040.901}
SPL {X  -159.990, Y  +466.881, Z    +0.000, E1   -23.322, E3 +472050.011}
SPL {X  -159.990, Y  +468.951, Z    +0.000, E1   -23.319, E3 +472060.203}
SPL {X  -159.990, Y  +471.818, Z    +0.000, E1   -23.351, E3 +472074.249}
SPL {X  -159.990, Y  +474.801, Z    +0.000, E1   -23.320, E3 +472089.025}
SPL {X  -159.990, Y  +476.830, Z    +0.000, E1   -23.323, E3 +472099.004}
SPL {X  -159.990, Y  +479.553, Z    +0.000, E1   -23.328, E3 +472112.407}
SPL {X  -159.990, Y  +482.950, Z    +0.000, E1   -23.350, E3 +472129.079}
SPL {X  -159.990, Y  +486.109, Z    +0.000, E1   -23.322, E3 +472144.694}
SPL {X  -159.990, Y  +488.481, Z    +0.000, E1   -23.319, E3 +472156.374}
SPL {X  -159.990, Y  +491.454, Z    +0.000, E1   -23.343, E3 +472170.954}
SPL {X  -159.990, Y  +494.937, Z    +0.000, E1   -23.343, E3 +472188.098}
SPL {X  -159.990, Y  +497.668, Z    +0.000, E1   -23.317, E3 +472201.591}
SPL {X  -159.990, Y  +499.995, Z    +0.000, E1   -23.324, E3 +472213.029}
SPL {X  -159.990, Y  +502.456, Z    +0.000, E1   -23.324, E3 +472225.144}
SPL {X  -159.990, Y  +505.646, Z    +0.000, E1   -23.350, E3 +472240.799}
SPL {X  -159.990, Y  +508.862, Z    +0.000, E1   -23.328, E3 +472256.664}
SPL {X  -159.990, Y  +510.971, Z    +0.000, E1   -23.308, E3 +472267.091}
SPL {X  -159.990, Y  +513.289, Z    +0.000, E1   -23.332, E3 +472278.458}
SPL {X  -159.990, Y  +516.860, Z    +0.000, E1   -23.355, E3 +472295.975}
SPL {X  -159.990, Y  +520.719, Z    +0.000, E1   -23.363, E3 +472314.886}
SPL {X  -159.990, Y  +523.968, Z    +0.000, E1   -23.332, E3 +472330.970}
SPL {X  -159.990, Y  +526.466, Z    +0.000, E1   -23.320, E3 +472343.314}
SPL {X  -159.990, Y  +528.815, Z    +0.000, E1   -23.322, E3 +472354.873}
SPL {X  -159.990, Y  +531.246, Z    +0.000, E1   -23.325, E3 +472366.812}
SPL {X  -159.990, Y  +534.143, Z    +0.000, E1   -23.341, E3 +472381.047}
SPL {X  -159.990, Y  +537.024, Z    +0.000, E1   -23.321, E3 +472395.290}
SPL {X  -159.990, Y  +539.129, Z    +0.000, E1   -23.310, E3 +472405.673}
SPL {X  -159.990, Y  +541.882, Z    +0.000, E1   -23.346, E3 +472419.154}
SPL {X  -159.990, Y  +544.941, Z    +0.000, E1   -23.325, E3 +472434.237}
SPL {X  -159.990, Y  +547.390, Z    +0.000, E1   -23.325, E3 +472446.290}
SPL {X  -159.990, Y  +550.708, Z    +0.000, E1   -23.357, E3 +472462.557}
SPL {X  -159.990, Y  +553.642, Z    +0.000, E1   -23.319, E3 +472477.064}
SPL {X  -159.990, Y  +555.637, Z    +0.000, E1   -23.323, E3 +472486.878}
SPL {X  -159.990, Y  +558.758, Z    +0.000, E1   -23.351, E3 +472502.188}
SPL {X  -159.990, Y  +561.830, Z    +0.000, E1   -23.325, E3 +472517.361}
SPL {X  -159.990, Y  +564.273, Z    +0.000, E1   -23.325, E3 +472529.386}
SPL {X  -159.990, Y  +567.351, Z    +0.000, E1   -23.348, E3 +472544.481}
SPL {X  -159.990, Y  +570.560, Z    +0.000, E1   -23.333, E3 +472560.311}
SPL {X  -159.990, Y  +572.975, Z    +0.000, E1   -23.316, E3 +472572.230}
SPL {X  -159.990, Y  +575.097, Z    +0.000, E1   -23.325, E3 +472582.657}
SPL {X  -159.990, Y  +578.356, Z    +0.000, E1   -23.358, E3 +472598.629}
SPL {X  -159.990, Y  +582.292, Z    +0.000, E1   -23.360, E3 +472617.945}
SPL {X  -159.990, Y  +585.165, Z    +0.000, E1   -23.322, E3 +472632.188}
SPL {X  -159.990, Y  +587.388, Z    +0.000, E1   -23.328, E3 +472643.101}
SPL {X  -159.990, Y  +589.763, Z    +0.000, E1   -23.328, E3 +472654.788}
SPL {X  -159.990, Y  +592.397, Z    +0.000, E1   -23.344, E3 +472667.668}
SPL {X  -159.990, Y  +595.589, Z    +0.000, E1   -23.356, E3 +472683.341}
SPL {X  -159.990, Y  +598.571, Z    +0.000, E1   -23.347, E3 +472697.985}
SPL {X  -159.990, Y  +600.935, Z    +0.000, E1   -23.343, E3 +472709.578}
SPL {X  -159.990, Y  +603.047, Z    +0.000, E1   -23.344, E3 +472719.964}
SPL {X  -159.990, Y  +605.187, Z    +0.000, E1   -23.344, E3 +472730.485}
SPL {X  -159.990, Y  +607.319, Z    +0.000, E1   -23.353, E3 +472740.948}
SPL {X  -159.990, Y  +609.514, Z    +0.000, E1   -23.337, E3 +472751.777}
SPL {X  -159.990, Y  +611.376, Z    +0.000, E1   -23.336, E3 +472760.964}
SPL {X  -159.990, Y  +613.591, Z    +0.000, E1   -23.342, E3 +472771.841}
SPL {X  -159.990, Y  +615.604, Z    +0.000, E1   -23.330, E3 +472781.779}
SPL {X  -159.990, Y  +617.623, Z    +0.000, E1   -23.337, E3 +472791.709}
SPL {X  -159.990, Y  +620.788, Z    +0.000, E1   -23.368, E3 +472807.215}
SPL {X  -159.990, Y  +623.764, Z    +0.000, E1   -23.335, E3 +472821.907}
SPL {X  -159.990, Y  +625.941, Z    +0.000, E1   -23.337, E3 +472832.598}
SPL {X  -159.990, Y  +628.611, Z    +0.000, E1   -23.357, E3 +472845.677}
SPL {X  -159.990, Y  +631.169, Z    +0.000, E1   -23.338, E3 +472858.281}
SPL {X  -159.990, Y  +633.318, Z    +0.000, E1   -23.339, E3 +472868.871}
SPL {X  -159.990, Y  +635.650, Z    +0.000, E1   -23.339, E3 +472880.341}
SPL {X  -159.990, Y  +637.839, Z    +0.000, E1   -23.335, E3 +472891.152}
SPL {X  -159.990, Y  +640.072, Z    +0.000, E1   -23.325, E3 +472902.184}
SPL {X  -159.990, Y  +642.230, Z    +0.000, E1   -23.323, E3 +472912.865}
SPL {X  -159.990, Y  +645.287, Z    +0.000, E1   -23.340, E3 +472927.891}
SPL {X  -159.990, Y  +647.803, Z    +0.000, E1   -23.310, E3 +472940.368}
SPL {X  -159.990, Y  +650.790, Z    +0.000, E1   -23.346, E3 +472954.976}
SPL {X  -159.990, Y  +654.543, Z    +0.000, E1   -23.348, E3 +472973.429}
SPL {X  -159.990, Y  +658.319, Z    +0.000, E1   -23.349, E3 +472992.018}
SPL {X  -159.990, Y  +661.392, Z    +0.000, E1   -23.318, E3 +473007.221}
SPL {X  -159.990, Y  +663.662, Z    +0.000, E1   -23.322, E3 +473018.345}
SPL {X  -159.990, Y  +665.964, Z    +0.000, E1   -23.328, E3 +473029.636}
SPL {X  -159.990, Y  +667.870, Z    +0.000, E1   -23.320, E3 +473039.043}
SPL {X  -159.990, Y  +669.861, Z    +0.000, E1   -23.321, E3 +473048.844}
SPL {X  -159.983, Y  +672.946, Z    +0.000, E1   -23.359, E3 +473063.953}
SPL {X  -159.924, Y  +676.110, Z    +0.000, E1   -23.320, E3 +473079.652}
SPL {X  -159.845, Y  +678.302, Z    +0.000, E1   -23.298, E3 +473090.554}
SPL {X  -159.760, Y  +680.081, Z    +0.000, E1   -23.288, E3 +473099.398}
SPL {X  -159.626, Y  +682.287, Z    +0.000, E1   -23.280, E3 +473110.369}
SPL {X  -159.462, Y  +684.486, Z    +0.000, E1   -23.258, E3 +473121.369}
SPL {X  -159.246, Y  +686.911, Z    +0.000, E1   -23.230, E3 +473133.530}
SPL {X  -159.019, Y  +689.098, Z    +0.000, E1   -23.200, E3 +473144.532}
SPL {X  -158.660, Y  +692.086, Z    +0.000, E1   -23.176, E3 +473159.576}
ENDSPLINE

SPLINE
SPL {X  -159.063, Y  +688.696, Z    +0.000, E1   -17.094, E3 +473201.858}
SPL {X  -159.987, Y  +672.488, Z    +0.000, E1    -5.638, E3 +473225.923}
SPL {X  -159.990, Y  +663.928, Z    +0.000, E1    +0.338, E3 +473231.717}
SPL {X  -159.990, Y  +658.009, Z    +0.000, E1    +4.774, E3 +473235.417}
SPL {X  -159.990, Y  +651.567, Z    +0.000, E1    +9.674, E3 +473240.821}
SPL {X  -159.990, Y  +638.711, Z    +0.000, E1   +17.883, E3 +473256.466}
SPL {X  -159.990, Y  +631.642, Z    +0.000, E1   +20.884, E3 +473272.025}
SPL {X  -159.990, Y  +626.048, Z    +0.000, E1   +22.026, E3 +473292.018}
SPL {X  -159.990, Y  +623.760, Z    +0.000, E1   +22.031, E3 +473304.005}
SPL {X  -159.990, Y  +621.334, Z    +0.000, E1   +22.029, E3 +473316.732}
SPL {X  -159.990, Y  +618.387, Z    +0.000, E1   +22.057, E3 +473332.122}
SPL {X  -159.990, Y  +615.830, Z    +0.000, E1   +22.023, E3 +473345.613}
SPL {X  -159.990, Y  +613.034, Z    +0.000, E1   +22.053, E3 +473360.220}
SPL {X  -159.990, Y  +609.503, Z    +0.000, E1   +22.054, E3 +473378.747}
SPL {X  -159.990, Y  +606.481, Z    +0.000, E1   +22.033, E3 +473394.621}
SPL {X  -159.990, Y  +603.419, Z    +0.000, E1   +22.064, E3 +473410.560}
SPL {X  -159.990, Y  +600.642, Z    +0.000, E1   +22.032, E3 +473425.190}
SPL {X  -159.990, Y  +598.568, Z    +0.000, E1   +22.046, E3 +473435.983}
SPL {X  -159.990, Y  +595.493, Z    +0.000, E1   +22.070, E3 +473452.066}
SPL {X  -159.990, Y  +592.865, Z    +0.000, E1   +22.036, E3 +473465.894}
SPL {X  -159.990, Y  +590.803, Z    +0.000, E1   +22.046, E3 +473476.685}
SPL {X  -159.990, Y  +587.778, Z    +0.000, E1   +22.073, E3 +473492.460}
SPL {X  -159.990, Y  +585.120, Z    +0.000, E1   +22.045, E3 +473506.404}
SPL {X  -159.990, Y  +583.118, Z    +0.000, E1   +22.052, E3 +473516.891}
SPL {X  -159.990, Y  +580.131, Z    +0.000, E1   +22.078, E3 +473532.497}
SPL {X  -159.990, Y  +576.888, Z    +0.000, E1   +22.061, E3 +473549.527}
SPL {X  -159.990, Y  +574.280, Z    +0.000, E1   +22.051, E3 +473563.201}
SPL {X  -159.990, Y  +572.375, Z    +0.000, E1   +22.037, E3 +473573.239}
SPL {X  -159.990, Y  +569.881, Z    +0.000, E1   +22.067, E3 +473586.233}
SPL {X  -159.990, Y  +567.211, Z    +0.000, E1   +22.046, E3 +473600.261}
SPL {X  -159.990, Y  +565.039, Z    +0.000, E1   +22.047, E3 +473611.638}
SPL {X  -159.990, Y  +562.755, Z    +0.000, E1   +22.047, E3 +473623.623}
SPL {X  -159.990, Y  +560.652, Z    +0.000, E1   +22.038, E3 +473634.669}
SPL {X  -159.990, Y  +558.852, Z    +0.000, E1   +22.046, E3 +473644.040}
SPL {X  -159.990, Y  +556.672, Z    +0.000, E1   +22.055, E3 +473655.430}
SPL {X  -159.990, Y  +553.726, Z    +0.000, E1   +22.080, E3 +473670.792}
SPL {X  -159.990, Y  +550.886, Z    +0.000, E1   +22.056, E3 +473685.731}
SPL {X  -159.990, Y  +548.814, Z    +0.000, E1   +22.049, E3 +473696.577}
SPL {X  -159.990, Y  +546.122, Z    +0.000, E1   +22.088, E3 +473710.590}
SPL {X  -159.990, Y  +542.390, Z    +0.000, E1   +22.086, E3 +473730.172}
SPL {X  -159.990, Y  +539.341, Z    +0.000, E1   +22.056, E3 +473746.194}
SPL {X  -159.990, Y  +536.301, Z    +0.000, E1   +22.084, E3 +473762.048}
SPL {X  -159.990, Y  +533.389, Z    +0.000, E1   +22.057, E3 +473777.356}
SPL {X  -159.990, Y  +531.347, Z    +0.000, E1   +22.052, E3 +473788.057}
SPL {X  -159.990, Y  +529.626, Z    +0.000, E1   +22.051, E3 +473797.054}
SPL {X  -159.990, Y  +527.412, Z    +0.000, E1   +22.067, E3 +473808.606}
SPL {X  -159.990, Y  +524.425, Z    +0.000, E1   +22.078, E3 +473824.239}
SPL {X  -159.990, Y  +521.599, Z    +0.000, E1   +22.060, E3 +473839.081}
SPL {X  -159.990, Y  +519.209, Z    +0.000, E1   +22.063, E3 +473851.556}
SPL {X  -159.990, Y  +516.651, Z    +0.000, E1   +22.071, E3 +473864.935}
SPL {X  -159.990, Y  +514.122, Z    +0.000, E1   +22.061, E3 +473878.207}
SPL {X  -159.990, Y  +511.670, Z    +0.000, E1   +22.064, E3 +473891.057}
SPL {X  -159.990, Y  +506.947, Z    +0.000, E1   +23.726, E3 +473901.086}
SPL {X  -159.990, Y  +496.921, Z    +0.000, E1   +28.340, E3 +473909.834}
SPL {X  -159.990, Y  +495.822, Z    +0.000, E1   +27.449, E3 +473920.582}
SPL {X  -159.990, Y  +494.952, Z    +0.000, E1   +26.628, E3 +473930.165}
SPL {X  -159.990, Y  +493.896, Z    +0.000, E1   +25.736, E3 +473941.495}
SPL {X  -159.990, Y  +491.647, Z    +0.000, E1   +25.401, E3 +473954.031}
SPL {X  -159.990, Y  +488.807, Z    +0.000, E1   +25.397, E3 +473966.729}
SPL {X  -159.990, Y  +486.070, Z    +0.000, E1   +25.399, E3 +473978.960}
SPL {X  -159.990, Y  +482.821, Z    +0.000, E1   +25.411, E3 +473993.461}
SPL {X  -159.990, Y  +480.183, Z    +0.000, E1   +25.384, E3 +474005.302}
SPL {X  -159.990, Y  +478.407, Z    +0.000, E1   +25.384, E3 +474013.242}
SPL {X  -159.990, Y  +475.940, Z    +0.000, E1   +25.403, E3 +474024.232}
SPL {X  -159.990, Y  +473.026, Z    +0.000, E1   +25.399, E3 +474037.262}
SPL {X  -159.990, Y  +470.047, Z    +0.000, E1   +25.402, E3 +474050.581}
SPL {X  -159.990, Y  +467.082, Z    +0.000, E1   +25.399, E3 +474063.828}
SPL {X  -159.990, Y  +464.919, Z    +0.000, E1   +25.381, E3 +474073.555}
SPL {X  -159.990, Y  +462.520, Z    +0.000, E1   +25.400, E3 +474084.229}
SPL {X  -159.990, Y  +460.081, Z    +0.000, E1   +25.390, E3 +474095.130}
SPL {X  -159.990, Y  +457.497, Z    +0.000, E1   +25.403, E3 +474106.655}
SPL {X  -159.990, Y  +454.323, Z    +0.000, E1   +25.412, E3 +474120.814}
SPL {X  -159.990, Y  +451.400, Z    +0.000, E1   +25.397, E3 +474133.905}
SPL {X  -159.990, Y  +448.503, Z    +0.000, E1   +25.410, E3 +474146.822}
SPL {X  -159.990, Y  +445.108, Z    +0.000, E1   +25.407, E3 +474162.060}
SPL {X  -159.990, Y  +441.797, Z    +0.000, E1   +25.390, E3 +474176.939}
SPL {X  -159.990, Y  +439.442, Z    +0.000, E1   +25.369, E3 +474187.517}
SPL {X  -159.990, Y  +436.316, Z    +0.000, E1   +25.420, E3 +474201.399}
SPL {X  -159.990, Y  +432.613, Z    +0.000, E1   +25.390, E3 +474218.024}
SPL {X  -159.990, Y  +429.079, Z    +0.000, E1   +25.407, E3 +474233.794}
SPL {X  -159.990, Y  +426.149, Z    +0.000, E1   +25.374, E3 +474246.956}
SPL {X  -159.990, Y  +423.417, Z    +0.000, E1   +25.400, E3 +474259.122}
SPL {X  -159.990, Y  +420.283, Z    +0.000, E1   +25.386, E3 +474273.166}
SPL {X  -159.990, Y  +417.514, Z    +0.000, E1   +25.386, E3 +474285.551}
SPL {X  -159.990, Y  +414.805, Z    +0.000, E1   +25.385, E3 +474297.671}
SPL {X  -159.990, Y  +411.282, Z    +0.000, E1   +25.413, E3 +474313.371}
SPL {X  -159.990, Y  +408.351, Z    +0.000, E1   +25.372, E3 +474326.558}
SPL {X  -159.990, Y  +405.773, Z    +0.000, E1   +25.398, E3 +474338.011}
SPL {X  -159.990, Y  +402.805, Z    +0.000, E1   +25.389, E3 +474351.297}
SPL {X  -159.990, Y  +400.083, Z    +0.000, E1   +25.388, E3 +474363.474}
SPL {X  -159.990, Y  +396.740, Z    +0.000, E1   +25.410, E3 +474378.398}
SPL {X  -159.990, Y  +392.622, Z    +0.000, E1   +25.413, E3 +474396.826}
SPL {X  -159.990, Y  +388.328, Z    +0.000, E1   +25.413, E3 +474416.054}
SPL {X  -159.990, Y  +384.900, Z    +0.000, E1   +25.383, E3 +474431.417}
SPL {X  -159.990, Y  +382.110, Z    +0.000, E1   +25.393, E3 +474443.863}
SPL {X  -159.961, Y  +379.439, Z    +0.000, E1   +25.380, E3 +474455.843}
SPL {X  -159.894, Y  +376.959, Z    +0.000, E1   +25.370, E3 +474467.020}
SPL {X  -159.784, Y  +374.382, Z    +0.000, E1   +25.356, E3 +474478.660}
SPL {X  -159.621, Y  +371.640, Z    +0.000, E1   +25.335, E3 +474491.100}
SPL {X  -159.406, Y  +368.844, Z    +0.000, E1   +25.307, E3 +474503.813}
SPL {X  -159.144, Y  +366.072, Z    +0.000, E1   +25.281, E3 +474516.421}
SPL {X  -158.822, Y  +363.200, Z    +0.000, E1   +25.236, E3 +474529.594}
SPL {X  -158.491, Y  +360.654, Z    +0.000, E1   +25.188, E3 +474541.334}
SPL {X  -158.127, Y  +358.155, Z    +0.000, E1   +25.126, E3 +474552.953}
SPL {X  -158.095, Y  +357.947, Z    +0.000, E1   +21.741, E3 +474584.525}
ENDSPLINE

SPLINE
SPL {X  -158.454, Y  +360.384, Z    +0.000, E1   +19.366, E3 +474596.677}
SPL {X  -159.737, Y  +373.507, Z    +0.000, E1   +10.311, E3 +474618.712}
SPL {X  -159.990, Y  +382.574, Z    +0.000, E1    +4.463, E3 +474625.400}
SPL {X  -159.990, Y  +389.909, Z    +0.000, E1    -0.662, E3 +474629.414}
SPL {X  -159.990, Y  +396.289, Z    +0.000, E1    -5.500, E3 +474633.194}
SPL {X  -159.990, Y  +407.941, Z    +0.000, E1   -14.126, E3 +474644.531}
SPL {X  -159.990, Y  +418.671, Z    +0.000, E1   -19.855, E3 +474663.948}
SPL {X  -159.990, Y  +428.534, Z    +0.000, E1   -23.299, E3 +474687.468}
SPL {X  -159.990, Y  +430.313, Z    +0.000, E1   -23.313, E3 +474696.181}
SPL {X  -159.990, Y  +432.766, Z    +0.000, E1   -23.321, E3 +474708.225}
SPL {X  -159.990, Y  +434.794, Z    +0.000, E1   -23.304, E3 +474718.256}
SPL {X  -159.990, Y  +437.007, Z    +0.000, E1   -23.323, E3 +474729.109}
SPL {X  -159.990, Y  +439.778, Z    +0.000, E1   -23.323, E3 +474742.741}
SPL {X  -159.990, Y  +442.010, Z    +0.000, E1   -23.308, E3 +474753.762}
SPL {X  -159.990, Y  +443.729, Z    +0.000, E1   -23.310, E3 +474762.219}
SPL {X  -159.990, Y  +446.037, Z    +0.000, E1   -23.324, E3 +474773.556}
SPL {X  -159.990, Y  +449.434, Z    +0.000, E1   -23.356, E3 +474790.177}
SPL {X  -159.990, Y  +452.308, Z    +0.000, E1   -23.313, E3 +474804.430}
SPL {X  -159.990, Y  +455.185, Z    +0.000, E1   -23.350, E3 +474818.494}
SPL {X  -159.990, Y  +458.265, Z    +0.000, E1   -23.328, E3 +474833.681}
SPL {X  -159.990, Y  +460.492, Z    +0.000, E1   -23.317, E3 +474844.680}
SPL {X  -159.990, Y  +462.929, Z    +0.000, E1   -23.331, E3 +474856.635}
SPL {X  -159.990, Y  +465.027, Z    +0.000, E1   -23.313, E3 +474866.988}
SPL {X  -159.990, Y  +466.881, Z    +0.000, E1   -23.322, E3 +474876.098}
SPL {X  -159.990, Y  +468.951, Z    +0.000, E1   -23.319, E3 +474886.290}
SPL {X  -159.990, Y  +471.818, Z    +0.000, E1   -23.351, E3 +474900.336}
SPL {X  -159.990, Y  +474.801, Z    +0.000, E1   -23.320, E3 +474915.112}
SPL {X  -159.990, Y  +476.830, Z    +0.000, E1   -23.323, E3 +474925.091}
SPL {X  -159.990, Y  +479.553, Z    +0.000, E1   -23.328, E3 +474938.494}
SPL {X  -159.990, Y  +481.893, Z    +0.000, E1   -23.312, E3 +474950.043}
SPL {X  -159.990, Y  +483.782, Z    +0.000, E1   -23.316, E3 +474959.329}
SPL {X  -159.990, Y  +486.109, Z    +0.000, E1   -23.322, E3 +474970.781}
SPL {X  -159.990, Y  +489.247, Z    +0.000, E1   -23.348, E3 +474986.169}
SPL {X  -159.990, Y  +493.031, Z    +0.000, E1   -23.350, E3 +475004.793}
SPL {X  -159.990, Y  +496.869, Z    +0.000, E1   -23.349, E3 +475023.683}
SPL {X  -159.990, Y  +499.995, Z    +0.000, E1   -23.324, E3 +475039.116}
SPL {X  -159.990, Y  +502.456, Z    +0.000, E1   -23.324, E3 +475051.231}
SPL {X  -159.990, Y  +505.646, Z    +0.000, E1   -23.350, E3 +475066.886}
SPL {X  -159.990, Y  +508.862, Z    +0.000, E1   -23.328, E3 +475082.751}
SPL {X  -159.990, Y  +510.971, Z    +0.000, E1   -23.308, E3 +475093.178}
SPL {X  -159.990, Y  +512.484, Z    +0.000, E1   -23.309, E3 +475100.628}
SPL {X  -159.990, Y  +514.757, Z    +0.000, E1   -23.329, E3 +475111.780}
SPL {X  -159.990, Y  +517.536, Z    +0.000, E1   -23.326, E3 +475125.447}
SPL {X  -159.990, Y  +519.961, Z    +0.000, E1   -23.334, E3 +475137.299}
SPL {X  -159.990, Y  +521.849, Z    +0.000, E1   -23.320, E3 +475146.621}
SPL {X  -159.990, Y  +523.968, Z    +0.000, E1   -23.332, E3 +475157.057}
SPL {X  -159.990, Y  +526.466, Z    +0.000, E1   -23.320, E3 +475169.401}
SPL {X  -159.990, Y  +528.815, Z    +0.000, E1   -23.322, E3 +475180.960}
SPL {X  -159.990, Y  +531.246, Z    +0.000, E1   -23.325, E3 +475192.899}
SPL {X  -159.990, Y  +533.354, Z    +0.000, E1   -23.318, E3 +475203.284}
SPL {X  -159.990, Y  +534.931, Z    +0.000, E1   -23.312, E3 +475211.079}
SPL {X  -159.990, Y  +537.024, Z    +0.000, E1   -23.321, E3 +475221.377}
SPL {X  -159.990, Y  +539.129, Z    +0.000, E1   -23.310, E3 +475231.760}
SPL {X  -159.990, Y  +541.183, Z    +0.000, E1   -23.319, E3 +475241.857}
SPL {X  -159.990, Y  +544.314, Z    +0.000, E1   -23.352, E3 +475257.185}
SPL {X  -159.990, Y  +548.126, Z    +0.000, E1   -23.354, E3 +475275.940}
SPL {X  -159.990, Y  +551.344, Z    +0.000, E1   -23.327, E3 +475291.832}
SPL {X  -159.990, Y  +553.642, Z    +0.000, E1   -23.319, E3 +475303.151}
SPL {X  -159.990, Y  +556.481, Z    +0.000, E1   -23.354, E3 +475317.058}
SPL {X  -159.990, Y  +559.475, Z    +0.000, E1   -23.321, E3 +475331.864}
SPL {X  -159.990, Y  +561.830, Z    +0.000, E1   -23.325, E3 +475343.448}
SPL {X  -159.990, Y  +564.273, Z    +0.000, E1   -23.325, E3 +475355.473}
SPL {X  -159.990, Y  +566.342, Z    +0.000, E1   -23.314, E3 +475365.677}
SPL {X  -159.990, Y  +568.184, Z    +0.000, E1   -23.317, E3 +475374.738}
SPL {X  -159.990, Y  +570.560, Z    +0.000, E1   -23.333, E3 +475386.398}
SPL {X  -159.990, Y  +572.975, Z    +0.000, E1   -23.316, E3 +475398.317}
SPL {X  -159.990, Y  +575.097, Z    +0.000, E1   -23.325, E3 +475408.744}
SPL {X  -159.990, Y  +578.356, Z    +0.000, E1   -23.358, E3 +475424.716}
SPL {X  -159.990, Y  +582.292, Z    +0.000, E1   -23.360, E3 +475444.032}
SPL {X  -159.990, Y  +585.165, Z    +0.000, E1   -23.322, E3 +475458.275}
SPL {X  -159.990, Y  +587.388, Z    +0.000, E1   -23.328, E3 +475469.187}
SPL {X  -159.990, Y  +590.594, Z    +0.000, E1   -23.363, E3 +475484.879}
SPL {X  -159.990, Y  +593.168, Z    +0.000, E1   -23.322, E3 +475497.592}
SPL {X  -159.990, Y  +595.589, Z    +0.000, E1   -23.356, E3 +475509.428}
SPL {X  -159.990, Y  +598.571, Z    +0.000, E1   -23.347, E3 +475524.072}
SPL {X  -159.990, Y  +600.935, Z    +0.000, E1   -23.343, E3 +475535.665}
SPL {X  -159.990, Y  +603.047, Z    +0.000, E1   -23.344, E3 +475546.051}
SPL {X  -159.990, Y  +605.187, Z    +0.000, E1   -23.344, E3 +475556.572}
SPL {X  -159.990, Y  +607.319, Z    +0.000, E1   -23.353, E3 +475567.035}
SPL {X  -159.990, Y  +609.514, Z    +0.000, E1   -23.337, E3 +475577.864}
SPL {X  -159.990, Y  +611.376, Z    +0.000, E1   -23.336, E3 +475587.051}
SPL {X  -159.990, Y  +613.591, Z    +0.000, E1   -23.342, E3 +475597.928}
SPL {X  -159.990, Y  +615.604, Z    +0.000, E1   -23.330, E3 +475607.866}
SPL {X  -159.990, Y  +617.623, Z    +0.000, E1   -23.337, E3 +475617.796}
SPL {X  -159.990, Y  +620.788, Z    +0.000, E1   -23.368, E3 +475633.302}
SPL {X  -159.990, Y  +623.764, Z    +0.000, E1   -23.335, E3 +475647.994}
SPL {X  -159.990, Y  +625.941, Z    +0.000, E1   -23.337, E3 +475658.685}
SPL {X  -159.990, Y  +628.611, Z    +0.000, E1   -23.357, E3 +475671.764}
SPL {X  -159.990, Y  +631.169, Z    +0.000, E1   -23.338, E3 +475684.368}
SPL {X  -159.990, Y  +633.318, Z    +0.000, E1   -23.339, E3 +475694.958}
SPL {X  -159.990, Y  +635.650, Z    +0.000, E1   -23.339, E3 +475706.428}
SPL {X  -159.990, Y  +637.839, Z    +0.000, E1   -23.335, E3 +475717.239}
SPL {X  -159.990, Y  +640.072, Z    +0.000, E1   -23.325, E3 +475728.271}
SPL {X  -159.990, Y  +642.230, Z    +0.000, E1   -23.323, E3 +475738.952}
SPL {X  -159.990, Y  +645.287, Z    +0.000, E1   -23.340, E3 +475753.978}
SPL {X  -159.990, Y  +647.803, Z    +0.000, E1   -23.310, E3 +475766.455}
SPL {X  -159.990, Y  +650.790, Z    +0.000, E1   -23.346, E3 +475781.063}
SPL {X  -159.990, Y  +654.543, Z    +0.000, E1   -23.348, E3 +475799.516}
SPL {X  -159.990, Y  +658.319, Z    +0.000, E1   -23.349, E3 +475818.105}
SPL {X  -159.990, Y  +661.392, Z    +0.000, E1   -23.318, E3 +475833.308}
SPL {X  -159.990, Y  +663.662, Z    +0.000, E1   -23.322, E3 +475844.432}
SPL {X  -159.990, Y  +665.964, Z    +0.000, E1   -23.328, E3 +475855.723}
SPL {X  -159.990, Y  +667.870, Z    +0.000, E1   -23.320, E3 +475865.130}
SPL {X  -159.990, Y  +669.861, Z    +0.000, E1   -23.321, E3 +475874.931}
SPL {X  -159.990, Y  +671.893, Z    +0.000, E1   -23.319, E3 +475884.939}
SPL {X  -159.974, Y  +673.789, Z    +0.000, E1   -23.323, E3 +475894.255}
SPL {X  -159.924, Y  +676.110, Z    +0.000, E1   -23.320, E3 +475905.739}
SPL {X  -159.801, Y  +679.265, Z    +0.000, E1   -23.327, E3 +475921.358}
SPL {X  -159.626, Y  +682.287, Z    +0.000, E1   -23.280, E3 +475936.456}
SPL {X  -159.462, Y  +684.486, Z    +0.000, E1   -23.258, E3 +475947.456}
SPL {X  -159.246, Y  +686.911, Z    +0.000, E1   -23.230, E3 +475959.617}
SPL {X  -159.019, Y  +689.098, Z    +0.000, E1   -23.200, E3 +475970.619}
SPL {X  -158.660, Y  +692.086, Z    +0.000, E1   -23.176, E3 +475985.663}
ENDSPLINE

SPLINE
SPL {X  -159.063, Y  +688.696, Z    +0.000, E1   -17.094, E3 +476027.945}
SPL {X  -159.967, Y  +674.206, Z    +0.000, E1    -6.731, E3 +476050.757}
SPL {X  -159.990, Y  +665.270, Z    +0.000, E1    -0.699, E3 +476056.927}
SPL {X  -159.990, Y  +658.009, Z    +0.000, E1    +4.774, E3 +476061.504}
SPL {X  -159.990, Y  +651.567, Z    +0.000, E1    +9.674, E3 +476066.907}
SPL {X  -159.990, Y  +638.711, Z    +0.000, E1   +17.883, E3 +476082.553}
SPL {X  -159.990, Y  +631.642, Z    +0.000, E1   +20.884, E3 +476098.112}
SPL {X  -159.990, Y  +626.048, Z    +0.000, E1   +22.026, E3 +476118.105}
SPL {X  -159.990, Y  +623.760, Z    +0.000, E1   +22.031, E3 +476130.092}
SPL {X  -159.990, Y  +621.334, Z    +0.000, E1   +22.029, E3 +476142.819}
SPL {X  -159.990, Y  +618.387, Z    +0.000, E1   +22.057, E3 +476158.209}
SPL {X  -159.990, Y  +614.928, Z    +0.000, E1   +22.055, E3 +476176.361}
SPL {X  -159.990, Y  +611.459, Z    +0.000, E1   +22.053, E3 +476194.564}
SPL {X  -159.990, Y  +608.810, Z    +0.000, E1   +22.023, E3 +476208.532}
SPL {X  -159.990, Y  +606.481, Z    +0.000, E1   +22.033, E3 +476220.708}
SPL {X  -159.990, Y  +603.419, Z    +0.000, E1   +22.064, E3 +476236.647}
SPL {X  -159.990, Y  +600.642, Z    +0.000, E1   +22.032, E3 +476251.277}
SPL {X  -159.990, Y  +598.568, Z    +0.000, E1   +22.046, E3 +476262.070}
SPL {X  -159.990, Y  +596.440, Z    +0.000, E1   +22.036, E3 +476273.251}
SPL {X  -159.990, Y  +593.768, Z    +0.000, E1   +22.071, E3 +476287.184}
SPL {X  -159.990, Y  +590.803, Z    +0.000, E1   +22.046, E3 +476302.772}
SPL {X  -159.990, Y  +587.778, Z    +0.000, E1   +22.073, E3 +476318.547}
SPL {X  -159.990, Y  +585.120, Z    +0.000, E1   +22.045, E3 +476332.491}
SPL {X  -159.990, Y  +583.118, Z    +0.000, E1   +22.052, E3 +476342.978}
SPL {X  -159.990, Y  +580.131, Z    +0.000, E1   +22.078, E3 +476358.584}
SPL {X  -159.990, Y  +576.888, Z    +0.000, E1   +22.061, E3 +476375.614}
SPL {X  -159.990, Y  +574.280, Z    +0.000, E1   +22.051, E3 +476389.288}
SPL {X  -159.990, Y  +572.375, Z    +0.000, E1   +22.037, E3 +476399.326}
SPL {X  -159.990, Y  +569.881, Z    +0.000, E1   +22.067, E3 +476412.320}
SPL {X  -159.990, Y  +567.211, Z    +0.000, E1   +22.046, E3 +476426.348}
SPL {X  -159.990, Y  +565.039, Z    +0.000, E1   +22.047, E3 +476437.725}
SPL {X  -159.990, Y  +562.755, Z    +0.000, E1   +22.047, E3 +476449.710}
SPL {X  -159.990, Y  +559.661, Z    +0.000, E1   +22.078, E3 +476465.842}
SPL {X  -159.990, Y  +555.965, Z    +0.000, E1   +22.085, E3 +476485.151}
SPL {X  -159.990, Y  +553.115, Z    +0.000, E1   +22.054, E3 +476500.137}
SPL {X  -159.990, Y  +550.886, Z    +0.000, E1   +22.056, E3 +476511.818}
SPL {X  -159.990, Y  +547.986, Z    +0.000, E1   +22.078, E3 +476526.937}
SPL {X  -159.990, Y  +545.350, Z    +0.000, E1   +22.053, E3 +476540.799}
SPL {X  -159.990, Y  +543.405, Z    +0.000, E1   +22.048, E3 +476551.012}
SPL {X  -159.990, Y  +541.673, Z    +0.000, E1   +22.053, E3 +476560.075}
SPL {X  -159.990, Y  +539.341, Z    +0.000, E1   +22.056, E3 +476572.281}
SPL {X  -159.990, Y  +536.301, Z    +0.000, E1   +22.084, E3 +476588.135}
SPL {X  -159.990, Y  +533.389, Z    +0.000, E1   +22.057, E3 +476603.443}
SPL {X  -159.990, Y  +531.347, Z    +0.000, E1   +22.052, E3 +476614.143}
SPL {X  -159.990, Y  +529.626, Z    +0.000, E1   +22.051, E3 +476623.141}
SPL {X  -159.990, Y  +527.412, Z    +0.000, E1   +22.067, E3 +476634.693}
SPL {X  -159.990, Y  +524.425, Z    +0.000, E1   +22.078, E3 +476650.326}
SPL {X  -159.990, Y  +521.599, Z    +0.000, E1   +22.060, E3 +476665.168}
SPL {X  -159.990, Y  +519.209, Z    +0.000, E1   +22.063, E3 +476677.643}
SPL {X  -159.990, Y  +516.651, Z    +0.000, E1   +22.071, E3 +476691.022}
SPL {X  -159.990, Y  +514.122, Z    +0.000, E1   +22.061, E3 +476704.294}
SPL {X  -159.990, Y  +511.670, Z    +0.000, E1   +22.064, E3 +476717.144}
SPL {X  -159.990, Y  +506.947, Z    +0.000, E1   +23.726, E3 +476727.173}
SPL {X  -159.990, Y  +496.921, Z    +0.000, E1   +28.340, E3 +476735.921}
SPL {X  -159.990, Y  +495.822, Z    +0.000, E1   +27.449, E3 +476746.669}
SPL {X  -159.990, Y  +494.952, Z    +0.000, E1   +26.628, E3 +476756.252}
SPL {X  -159.990, Y  +493.896, Z    +0.000, E1   +25.736, E3 +476767.582}
SPL {X  -159.990, Y  +491.647, Z    +0.000, E1   +25.401, E3 +476780.118}
SPL {X  -159.990, Y  +488.807, Z    +0.000, E1   +25.397, E3 +476792.816}
SPL {X  -159.990, Y  +486.070, Z    +0.000, E1   +25.399, E3 +476805.047}
SPL {X  -159.990, Y  +483.747, Z    +0.000, E1   +25.384, E3 +476815.460}
SPL {X  -159.990, Y  +481.980, Z    +0.000, E1   +25.384, E3 +476823.358}
SPL {X  -159.990, Y  +479.252, Z    +0.000, E1   +25.412, E3 +476835.499}
SPL {X  -159.990, Y  +475.940, Z    +0.000, E1   +25.403, E3 +476850.319}
SPL {X  -159.990, Y  +473.026, Z    +0.000, E1   +25.399, E3 +476863.349}
SPL {X  -159.990, Y  +470.047, Z    +0.000, E1   +25.402, E3 +476876.668}
SPL {X  -159.990, Y  +466.213, Z    +0.000, E1   +25.433, E3 +476893.747}
SPL {X  -159.990, Y  +462.520, Z    +0.000, E1   +25.400, E3 +476910.316}
SPL {X  -159.990, Y  +460.081, Z    +0.000, E1   +25.390, E3 +476921.217}
SPL {X  -159.990, Y  +457.497, Z    +0.000, E1   +25.403, E3 +476932.742}
SPL {X  -159.990, Y  +455.126, Z    +0.000, E1   +25.389, E3 +476943.350}
SPL {X  -159.990, Y  +452.123, Z    +0.000, E1   +25.426, E3 +476956.708}
SPL {X  -159.990, Y  +448.503, Z    +0.000, E1   +25.410, E3 +476972.909}
SPL {X  -159.990, Y  +445.882, Z    +0.000, E1   +25.385, E3 +476984.712}
SPL {X  -159.990, Y  +443.345, Z    +0.000, E1   +25.390, E3 +476996.094}
SPL {X  -159.990, Y  +441.077, Z    +0.000, E1   +25.369, E3 +477006.292}
SPL {X  -159.990, Y  +438.608, Z    +0.000, E1   +25.392, E3 +477017.289}
SPL {X  -159.990, Y  +434.852, Z    +0.000, E1   +25.415, E3 +477034.044}
SPL {X  -159.990, Y  +430.645, Z    +0.000, E1   +25.414, E3 +477052.863}
SPL {X  -159.990, Y  +426.865, Z    +0.000, E1   +25.398, E3 +477069.793}
SPL {X  -159.990, Y  +424.251, Z    +0.000, E1   +25.375, E3 +477081.530}
SPL {X  -159.990, Y  +421.010, Z    +0.000, E1   +25.418, E3 +477095.945}
SPL {X  -159.990, Y  +417.514, Z    +0.000, E1   +25.386, E3 +477111.638}
SPL {X  -159.990, Y  +414.805, Z    +0.000, E1   +25.385, E3 +477123.758}
SPL {X  -159.990, Y  +411.282, Z    +0.000, E1   +25.413, E3 +477139.458}
SPL {X  -159.990, Y  +408.351, Z    +0.000, E1   +25.372, E3 +477152.645}
SPL {X  -159.990, Y  +405.773, Z    +0.000, E1   +25.398, E3 +477164.098}
SPL {X  -159.990, Y  +402.805, Z    +0.000, E1   +25.389, E3 +477177.384}
SPL {X  -159.990, Y  +400.083, Z    +0.000, E1   +25.388, E3 +477189.561}
SPL {X  -159.990, Y  +396.740, Z    +0.000, E1   +25.410, E3 +477204.485}
SPL {X  -159.990, Y  +392.622, Z    +0.000, E1   +25.413, E3 +477222.913}
SPL {X  -159.990, Y  +388.328, Z    +0.000, E1   +25.413, E3 +477242.141}
SPL {X  -159.990, Y  +384.900, Z    +0.000, E1   +25.383, E3 +477257.504}
SPL {X  -159.990, Y  +382.110, Z    +0.000, E1   +25.393, E3 +477269.950}
SPL {X  -159.961, Y  +379.439, Z    +0.000, E1   +25.380, E3 +477281.930}
SPL {X  -159.894, Y  +376.959, Z    +0.000, E1   +25.370, E3 +477293.107}
SPL {X  -159.784, Y  +374.382, Z    +0.000, E1   +25.356, E3 +477304.747}
SPL {X  -159.621, Y  +371.640, Z    +0.000, E1   +25.335, E3 +477317.187}
SPL {X  -159.406, Y  +368.844, Z    +0.000, E1   +25.307, E3 +477329.900}
SPL {X  -159.144, Y  +366.072, Z    +0.000, E1   +25.281, E3 +477342.508}
SPL {X  -158.822, Y  +363.200, Z    +0.000, E1   +25.236, E3 +477355.681}
SPL {X  -158.491, Y  +360.654, Z    +0.000, E1   +25.188, E3 +477367.421}
SPL {X  -158.127, Y  +358.155, Z    +0.000, E1   +25.126, E3 +477379.040}
SPL {X  -158.095, Y  +357.947, Z    +0.000, E1   +21.741, E3 +477410.612}
ENDSPLINE

SPLINE
SPL {X  -158.454, Y  +360.384, Z    +0.000, E1   +19.366, E3 +477422.764}
SPL {X  -159.737, Y  +373.507, Z    +0.000, E1   +10.311, E3 +477444.799}
SPL {X  -159.990, Y  +382.574, Z    +0.000, E1    +4.463, E3 +477451.487}
SPL {X  -159.990, Y  +387.496, Z    +0.000, E1    +1.004, E3 +477454.232}
SPL {X  -159.990, Y  +395.121, Z    +0.000, E1    -4.514, E3 +477458.544}
SPL {X  -159.990, Y  +407.941, Z    +0.000, E1   -14.126, E3 +477470.618}
SPL {X  -159.990, Y  +418.671, Z    +0.000, E1   -19.855, E3 +477490.035}
SPL {X  -159.990, Y  +428.534, Z    +0.000, E1   -23.299, E3 +477513.555}
SPL {X  -159.990, Y  +431.017, Z    +0.000, E1   -23.339, E3 +477525.681}
SPL {X  -159.990, Y  +434.188, Z    +0.000, E1   -23.325, E3 +477541.305}
SPL {X  -159.990, Y  +437.007, Z    +0.000, E1   -23.323, E3 +477555.196}
SPL {X  -159.990, Y  +439.778, Z    +0.000, E1   -23.323, E3 +477568.828}
SPL {X  -159.990, Y  +442.945, Z    +0.000, E1   -23.339, E3 +477584.392}
SPL {X  -159.990, Y  +446.037, Z    +0.000, E1   -23.324, E3 +477599.642}
SPL {X  -159.990, Y  +449.434, Z    +0.000, E1   -23.356, E3 +477616.264}
SPL {X  -159.990, Y  +452.308, Z    +0.000, E1   -23.313, E3 +477630.517}
SPL {X  -159.990, Y  +455.185, Z    +0.000, E1   -23.350, E3 +477644.581}
SPL {X  -159.990, Y  +458.265, Z    +0.000, E1   -23.328, E3 +477659.767}
SPL {X  -159.990, Y  +460.492, Z    +0.000, E1   -23.317, E3 +477670.767}
SPL {X  -159.990, Y  +462.929, Z    +0.000, E1   -23.331, E3 +477682.722}
SPL {X  -159.990, Y  +465.027, Z    +0.000, E1   -23.313, E3 +477693.075}
SPL {X  -159.990, Y  +466.881, Z    +0.000, E1   -23.322, E3 +477702.185}
SPL {X  -159.990, Y  +468.951, Z    +0.000, E1   -23.319, E3 +477712.377}
SPL {X  -159.990, Y  +471.818, Z    +0.000, E1   -23.351, E3 +477726.423}
SPL {X  -159.990, Y  +474.801, Z    +0.000, E1   -23.320, E3 +477741.199}
SPL {X  -159.990, Y  +476.830, Z    +0.000, E1   -23.323, E3 +477751.178}
SPL {X  -159.990, Y  +479.553, Z    +0.000, E1   -23.328, E3 +477764.580}
SPL {X  -159.990, Y  +482.950, Z    +0.000, E1   -23.350, E3 +477781.253}
SPL {X  -159.990, Y  +486.109, Z    +0.000, E1   -23.322, E3 +477796.868}
SPL {X  -159.990, Y  +488.481, Z    +0.000, E1   -23.319, E3 +477808.548}
SPL {X  -159.990, Y  +491.454, Z    +0.000, E1   -23.343, E3 +477823.128}
SPL {X  -159.990, Y  +494.937, Z    +0.000, E1   -23.343, E3 +477840.272}
SPL {X  -159.990, Y  +497.668, Z    +0.000, E1   -23.317, E3 +477853.765}
SPL {X  -159.990, Y  +499.995, Z    +0.000, E1   -23.324, E3 +477865.203}
SPL {X  -159.990, Y  +502.456, Z    +0.000, E1   -23.324, E3 +477877.318}
SPL {X  -159.990, Y  +504.508, Z    +0.000, E1   -23.311, E3 +477887.452}
SPL {X  -159.990, Y  +506.420, Z    +0.000, E1   -23.317, E3 +477896.845}
SPL {X  -159.990, Y  +508.862, Z    +0.000, E1   -23.328, E3 +477908.838}
SPL {X  -159.990, Y  +511.771, Z    +0.000, E1   -23.331, E3 +477923.159}
SPL {X  -159.990, Y  +514.757, Z    +0.000, E1   -23.329, E3 +477937.867}
SPL {X  -159.990, Y  +517.536, Z    +0.000, E1   -23.326, E3 +477951.534}
SPL {X  -159.990, Y  +520.719, Z    +0.000, E1   -23.363, E3 +477967.060}
SPL {X  -159.990, Y  +523.968, Z    +0.000, E1   -23.332, E3 +477983.144}
SPL {X  -159.990, Y  +526.466, Z    +0.000, E1   -23.320, E3 +477995.488}
SPL {X  -159.990, Y  +528.815, Z    +0.000, E1   -23.322, E3 +478007.047}
SPL {X  -159.990, Y  +531.246, Z    +0.000, E1   -23.325, E3 +478018.986}
SPL {X  -159.990, Y  +533.354, Z    +0.000, E1   -23.318, E3 +478029.371}
SPL {X  -159.990, Y  +534.931, Z    +0.000, E1   -23.312, E3 +478037.166}
SPL {X  -159.990, Y  +537.024, Z    +0.000, E1   -23.321, E3 +478047.464}
SPL {X  -159.990, Y  +539.129, Z    +0.000, E1   -23.310, E3 +478057.847}
SPL {X  -159.990, Y  +541.183, Z    +0.000, E1   -23.319, E3 +478067.944}
SPL {X  -159.990, Y  +544.314, Z    +0.000, E1   -23.352, E3 +478083.272}
SPL {X  -159.990, Y  +548.126, Z    +0.000, E1   -23.354, E3 +478102.027}
SPL {X  -159.990, Y  +551.344, Z    +0.000, E1   -23.327, E3 +478117.919}
SPL {X  -159.990, Y  +553.642, Z    +0.000, E1   -23.319, E3 +478129.238}
SPL {X  -159.990, Y  +556.481, Z    +0.000, E1   -23.354, E3 +478143.145}
SPL {X  -159.990, Y  +559.475, Z    +0.000, E1   -23.321, E3 +478157.951}
SPL {X  -159.990, Y  +561.830, Z    +0.000, E1   -23.325, E3 +478169.535}
SPL {X  -159.990, Y  +564.273, Z    +0.000, E1   -23.325, E3 +478181.560}
SPL {X  -159.990, Y  +566.342, Z    +0.000, E1   -23.314, E3 +478191.764}
SPL {X  -159.990, Y  +568.184, Z    +0.000, E1   -23.317, E3 +478200.825}
SPL {X  -159.990, Y  +570.560, Z    +0.000, E1   -23.333, E3 +478212.485}
SPL {X  -159.990, Y  +572.975, Z    +0.000, E1   -23.316, E3 +478224.404}
SPL {X  -159.990, Y  +575.097, Z    +0.000, E1   -23.325, E3 +478234.831}
SPL {X  -159.990, Y  +578.356, Z    +0.000, E1   -23.358, E3 +478250.803}
SPL {X  -159.990, Y  +582.292, Z    +0.000, E1   -23.360, E3 +478270.119}
SPL {X  -159.990, Y  +585.165, Z    +0.000, E1   -23.322, E3 +478284.362}
SPL {X  -159.990, Y  +587.388, Z    +0.000, E1   -23.328, E3 +478295.274}
SPL {X  -159.990, Y  +590.594, Z    +0.000, E1   -23.363, E3 +478310.966}
SPL {X  -159.990, Y  +594.301, Z    +0.000, E1   -23.358, E3 +478329.171}
SPL {X  -159.990, Y  +597.981, Z    +0.000, E1   -23.373, E3 +478347.219}
SPL {X  -159.990, Y  +600.935, Z    +0.000, E1   -23.343, E3 +478361.752}
SPL {X  -159.990, Y  +603.047, Z    +0.000, E1   -23.344, E3 +478372.137}
SPL {X  -159.990, Y  +605.187, Z    +0.000, E1   -23.344, E3 +478382.659}
SPL {X  -159.990, Y  +607.319, Z    +0.000, E1   -23.353, E3 +478393.122}
SPL {X  -159.990, Y  +610.569, Z    +0.000, E1   -23.372, E3 +478409.086}
SPL {X  -159.990, Y  +613.591, Z    +0.000, E1   -23.342, E3 +478424.015}
SPL {X  -159.990, Y  +615.604, Z    +0.000, E1   -23.330, E3 +478433.953}
SPL {X  -159.990, Y  +618.445, Z    +0.000, E1   -23.368, E3 +478447.866}
SPL {X  -159.990, Y  +621.517, Z    +0.000, E1   -23.337, E3 +478463.030}
SPL {X  -159.990, Y  +623.764, Z    +0.000, E1   -23.335, E3 +478474.081}
SPL {X  -159.990, Y  +626.608, Z    +0.000, E1   -23.361, E3 +478488.006}
SPL {X  -159.990, Y  +630.271, Z    +0.000, E1   -23.375, E3 +478505.967}
SPL {X  -159.990, Y  +633.318, Z    +0.000, E1   -23.339, E3 +478521.044}
SPL {X  -159.990, Y  +635.650, Z    +0.000, E1   -23.339, E3 +478532.515}
SPL {X  -159.990, Y  +637.839, Z    +0.000, E1   -23.335, E3 +478543.326}
SPL {X  -159.990, Y  +640.072, Z    +0.000, E1   -23.325, E3 +478554.358}
SPL {X  -159.990, Y  +643.026, Z    +0.000, E1   -23.354, E3 +478568.898}
SPL {X  -159.990, Y  +646.970, Z    +0.000, E1   -23.346, E3 +478588.361}
SPL {X  -159.990, Y  +650.790, Z    +0.000, E1   -23.346, E3 +478607.150}
SPL {X  -159.990, Y  +654.543, Z    +0.000, E1   -23.348, E3 +478625.603}
SPL {X  -159.990, Y  +658.319, Z    +0.000, E1   -23.349, E3 +478644.192}
SPL {X  -159.990, Y  +661.392, Z    +0.000, E1   -23.318, E3 +478659.395}
SPL {X  -159.990, Y  +663.662, Z    +0.000, E1   -23.322, E3 +478670.519}
SPL {X  -159.990, Y  +665.964, Z    +0.000, E1   -23.328, E3 +478681.810}
SPL {X  -159.990, Y  +667.870, Z    +0.000, E1   -23.320, E3 +478691.217}
SPL {X  -159.990, Y  +669.861, Z    +0.000, E1   -23.321, E3 +478701.018}
SPL {X  -159.990, Y  +671.893, Z    +0.000, E1   -23.319, E3 +478711.026}
SPL {X  -159.974, Y  +673.789, Z    +0.000, E1   -23.323, E3 +478720.342}
SPL {X  -159.924, Y  +676.110, Z    +0.000, E1   -23.320, E3 +478731.826}
SPL {X  -159.801, Y  +679.265, Z    +0.000, E1   -23.327, E3 +478747.445}
SPL {X  -159.626, Y  +682.287, Z    +0.000, E1   -23.280, E3 +478762.543}
SPL {X  -159.462, Y  +684.486, Z    +0.000, E1   -23.258, E3 +478773.543}
SPL {X  -159.246, Y  +686.911, Z    +0.000, E1   -23.230, E3 +478785.704}
SPL {X  -159.019, Y  +689.098, Z    +0.000, E1   -23.200, E3 +478796.706}
SPL {X  -158.660, Y  +692.086, Z    +0.000, E1   -23.176, E3 +478811.750}
ENDSPLINE

SPLINE
SPL {X  -159.063, Y  +688.696, Z    +0.000, E1   -17.094, E3 +478854.032}
SPL {X  -159.987, Y  +672.488, Z    +0.000, E1    -5.638, E3 +478878.097}
SPL {X  -159.990, Y  +663.928, Z    +0.000, E1    +0.338, E3 +478883.891}
SPL {X  -159.990, Y  +658.009, Z    +0.000, E1    +4.774, E3 +478887.591}
SPL {X  -159.990, Y  +651.567, Z    +0.000, E1    +9.674, E3 +478892.994}
SPL {X  -159.990, Y  +638.711, Z    +0.000, E1   +17.883, E3 +478908.640}
SPL {X  -159.990, Y  +631.642, Z    +0.000, E1   +20.884, E3 +478924.199}
SPL {X  -159.990, Y  +626.048, Z    +0.000, E1   +22.026, E3 +478944.192}
SPL {X  -159.990, Y  +623.760, Z    +0.000, E1   +22.031, E3 +478956.179}
SPL {X  -159.990, Y  +621.334, Z    +0.000, E1   +22.029, E3 +478968.906}
SPL {X  -159.990, Y  +618.387, Z    +0.000, E1   +22.057, E3 +478984.296}
SPL {X  -159.990, Y  +614.928, Z    +0.000, E1   +22.055, E3 +479002.448}
SPL {X  -159.990, Y  +611.459, Z    +0.000, E1   +22.053, E3 +479020.651}
SPL {X  -159.990, Y  +608.810, Z    +0.000, E1   +22.023, E3 +479034.619}
SPL {X  -159.990, Y  +606.481, Z    +0.000, E1   +22.033, E3 +479046.795}
SPL {X  -159.990, Y  +603.419, Z    +0.000, E1   +22.064, E3 +479062.734}
SPL {X  -159.990, Y  +600.642, Z    +0.000, E1   +22.032, E3 +479077.364}
SPL {X  -159.990, Y  +598.568, Z    +0.000, E1   +22.046, E3 +479088.156}
SPL {X  -159.990, Y  +595.493, Z    +0.000, E1   +22.070, E3 +479104.240}
SPL {X  -159.990, Y  +592.865, Z    +0.000, E1   +22.036, E3 +479118.068}
SPL {X  -159.990, Y  +590.803, Z    +0.000, E1   +22.046, E3 +479128.859}
SPL {X  -159.990, Y  +587.778, Z    +0.000, E1   +22.073, E3 +479144.634}
SPL {X  -159.990, Y  +585.120, Z    +0.000, E1   +22.045, E3 +479158.578}
SPL {X  -159.990, Y  +583.118, Z    +0.000, E1   +22.052, E3 +479169.064}
SPL {X  -159.990, Y  +580.131, Z    +0.000, E1   +22.078, E3 +479184.671}
SPL {X  -159.990, Y  +576.888, Z    +0.000, E1   +22.061, E3 +479201.701}
SPL {X  -159.990, Y  +574.280, Z    +0.000, E1   +22.051, E3 +479215.375}
SPL {X  -159.990, Y  +572.375, Z    +0.000, E1   +22.037, E3 +479225.413}
SPL {X  -159.990, Y  +569.881, Z    +0.000, E1   +22.067, E3 +479238.407}
SPL {X  -159.990, Y  +567.211, Z    +0.000, E1   +22.046, E3 +479252.435}
SPL {X  -159.990, Y  +565.039, Z    +0.000, E1   +22.047, E3 +479263.812}
SPL {X  -159.990, Y  +562.755, Z    +0.000, E1   +22.047, E3 +479275.797}
SPL {X  -159.990, Y  +559.661, Z    +0.000, E1   +22.078, E3 +479291.929}
SPL {X  -159.990, Y  +555.965, Z    +0.000, E1   +22.085, E3 +479311.238}
SPL {X  -159.990, Y  +553.115, Z    +0.000, E1   +22.054, E3 +479326.224}
SPL {X  -159.990, Y  +550.886, Z    +0.000, E1   +22.056, E3 +479337.905}
SPL {X  -159.990, Y  +547.986, Z    +0.000, E1   +22.078, E3 +479353.024}
SPL {X  -159.990, Y  +545.350, Z    +0.000, E1   +22.053, E3 +479366.886}
SPL {X  -159.990, Y  +543.405, Z    +0.000, E1   +22.048, E3 +479377.099}
SPL {X  -159.990, Y  +541.673, Z    +0.000, E1   +22.053, E3 +479386.162}
SPL {X  -159.990, Y  +539.341, Z    +0.000, E1   +22.056, E3 +479398.368}
SPL {X  -159.990, Y  +536.301, Z    +0.000, E1   +22.084, E3 +479414.222}
SPL {X  -159.990, Y  +533.389, Z    +0.000, E1   +22.057, E3 +479429.530}
SPL {X  -159.990, Y  +531.347, Z    +0.000, E1   +22.052, E3 +479440.230}
SPL {X  -159.990, Y  +529.626, Z    +0.000, E1   +22.051, E3 +479449.228}
SPL {X  -159.990, Y  +527.412, Z    +0.000, E1   +22.067, E3 +479460.780}
SPL {X  -159.990, Y  +524.425, Z    +0.000, E1   +22.078, E3 +479476.413}
SPL {X  -159.990, Y  +521.599, Z    +0.000, E1   +22.060, E3 +479491.255}
SPL {X  -159.990, Y  +519.209, Z    +0.000, E1   +22.063, E3 +479503.730}
SPL {X  -159.990, Y  +516.651, Z    +0.000, E1   +22.071, E3 +479517.109}
SPL {X  -159.990, Y  +514.122, Z    +0.000, E1   +22.061, E3 +479530.381}
SPL {X  -159.990, Y  +511.670, Z    +0.000, E1   +22.064, E3 +479543.231}
SPL {X  -159.990, Y  +506.947, Z    +0.000, E1   +23.726, E3 +479553.260}
SPL {X  -159.990, Y  +496.921, Z    +0.000, E1   +28.340, E3 +479562.008}
SPL {X  -159.990, Y  +495.822, Z    +0.000, E1   +27.449, E3 +479572.756}
SPL {X  -159.990, Y  +494.952, Z    +0.000, E1   +26.628, E3 +479582.339}
SPL {X  -159.990, Y  +493.896, Z    +0.000, E1   +25.736, E3 +479593.669}
SPL {X  -159.990, Y  +491.647, Z    +0.000, E1   +25.401, E3 +479606.204}
SPL {X  -159.990, Y  +488.807, Z    +0.000, E1   +25.397, E3 +479618.903}
SPL {X  -159.990, Y  +486.070, Z    +0.000, E1   +25.399, E3 +479631.134}
SPL {X  -159.990, Y  +483.747, Z    +0.000, E1   +25.384, E3 +479641.547}
SPL {X  -159.990, Y  +481.038, Z    +0.000, E1   +25.412, E3 +479653.602}
SPL {X  -159.990, Y  +478.407, Z    +0.000, E1   +25.384, E3 +479665.416}
SPL {X  -159.990, Y  +475.940, Z    +0.000, E1   +25.403, E3 +479676.406}
SPL {X  -159.990, Y  +473.026, Z    +0.000, E1   +25.399, E3 +479689.436}
SPL {X  -159.990, Y  +470.047, Z    +0.000, E1   +25.402, E3 +479702.755}
SPL {X  -159.990, Y  +466.213, Z    +0.000, E1   +25.433, E3 +479719.834}
SPL {X  -159.990, Y  +462.520, Z    +0.000, E1   +25.400, E3 +479736.403}
SPL {X  -159.990, Y  +460.081, Z    +0.000, E1   +25.390, E3 +479747.304}
SPL {X  -159.990, Y  +457.497, Z    +0.000, E1   +25.403, E3 +479758.829}
SPL {X  -159.990, Y  +455.126, Z    +0.000, E1   +25.389, E3 +479769.437}
SPL {X  -159.990, Y  +453.438, Z    +0.000, E1   +25.385, E3 +479776.997}
SPL {X  -159.990, Y  +450.823, Z    +0.000, E1   +25.417, E3 +479788.617}
SPL {X  -159.990, Y  +446.894, Z    +0.000, E1   +25.428, E3 +479806.174}
SPL {X  -159.990, Y  +443.345, Z    +0.000, E1   +25.390, E3 +479822.181}
SPL {X  -159.990, Y  +441.077, Z    +0.000, E1   +25.369, E3 +479832.379}
SPL {X  -159.990, Y  +438.608, Z    +0.000, E1   +25.392, E3 +479843.376}
SPL {X  -159.990, Y  +434.852, Z    +0.000, E1   +25.415, E3 +479860.131}
SPL {X  -159.990, Y  +431.966, Z    +0.000, E1   +25.371, E3 +479873.128}
SPL {X  -159.990, Y  +429.079, Z    +0.000, E1   +25.407, E3 +479885.968}
SPL {X  -159.990, Y  +426.149, Z    +0.000, E1   +25.374, E3 +479899.130}
SPL {X  -159.990, Y  +423.417, Z    +0.000, E1   +25.400, E3 +479911.296}
SPL {X  -159.990, Y  +420.283, Z    +0.000, E1   +25.386, E3 +479925.340}
SPL {X  -159.990, Y  +417.514, Z    +0.000, E1   +25.386, E3 +479937.725}
SPL {X  -159.990, Y  +414.805, Z    +0.000, E1   +25.385, E3 +479949.845}
SPL {X  -159.990, Y  +411.959, Z    +0.000, E1   +25.386, E3 +479962.571}
SPL {X  -159.990, Y  +408.981, Z    +0.000, E1   +25.392, E3 +479975.875}
SPL {X  -159.990, Y  +405.773, Z    +0.000, E1   +25.398, E3 +479990.185}
SPL {X  -159.990, Y  +402.805, Z    +0.000, E1   +25.389, E3 +480003.471}
SPL {X  -159.990, Y  +400.083, Z    +0.000, E1   +25.388, E3 +480015.648}
SPL {X  -159.990, Y  +396.740, Z    +0.000, E1   +25.410, E3 +480030.572}
SPL {X  -159.990, Y  +393.569, Z    +0.000, E1   +25.379, E3 +480044.822}
SPL {X  -159.990, Y  +390.564, Z    +0.000, E1   +25.393, E3 +480058.266}
SPL {X  -159.990, Y  +387.503, Z    +0.000, E1   +25.378, E3 +480071.981}
SPL {X  -159.990, Y  +384.900, Z    +0.000, E1   +25.383, E3 +480083.591}
SPL {X  -159.990, Y  +382.110, Z    +0.000, E1   +25.393, E3 +480096.037}
SPL {X  -159.961, Y  +379.439, Z    +0.000, E1   +25.380, E3 +480108.017}
SPL {X  -159.894, Y  +376.959, Z    +0.000, E1   +25.370, E3 +480119.194}
SPL {X  -159.784, Y  +374.382, Z    +0.000, E1   +25.356, E3 +480130.834}
SPL {X  -159.621, Y  +371.640, Z    +0.000, E1   +25.335, E3 +480143.274}
SPL {X  -159.406, Y  +368.844, Z    +0.000, E1   +25.307, E3 +480155.987}
SPL {X  -159.144, Y  +366.072, Z    +0.000, E1   +25.281, E3 +480168.595}
SPL {X  -158.822, Y  +363.200, Z    +0.000, E1   +25.236, E3 +480181.768}
SPL {X  -158.491, Y  +360.654, Z    +0.000, E1   +25.188, E3 +480193.508}
SPL {X  -158.127, Y  +358.155, Z    +0.000, E1   +25.126, E3 +480205.127}
SPL {X  -158.095, Y  +357.947, Z    +0.000, E1   +21.741, E3 +480236.699}
ENDSPLINE

SPLINE
SPL {X  -158.454, Y  +360.384, Z    +0.000, E1   +19.366, E3 +480248.851}
SPL {X  -159.737, Y  +373.507, Z    +0.000, E1   +10.311, E3 +480270.886}
SPL {X  -159.990, Y  +382.574, Z    +0.000, E1    +4.463, E3 +480277.574}
SPL {X  -159.990, Y  +387.496, Z    +0.000, E1    +1.004, E3 +480280.319}
SPL {X  -159.990, Y  +395.121, Z    +0.000, E1    -4.514, E3 +480284.631}
SPL {X  -159.990, Y  +407.941, Z    +0.000, E1   -14.126, E3 +480296.705}
SPL {X  -159.990, Y  +418.671, Z    +0.000, E1   -19.855, E3 +480316.122}
SPL {X  -159.990, Y  +429.878, Z    +0.000, E1   -23.330, E3 +480346.177}
SPL {X  -159.990, Y  +432.766, Z    +0.000, E1   -23.321, E3 +480360.399}
SPL {X  -159.990, Y  +434.794, Z    +0.000, E1   -23.304, E3 +480370.430}
SPL {X  -159.990, Y  +437.007, Z    +0.000, E1   -23.323, E3 +480381.283}
SPL {X  -159.990, Y  +439.778, Z    +0.000, E1   -23.323, E3 +480394.915}
SPL {X  -159.990, Y  +442.945, Z    +0.000, E1   -23.339, E3 +480410.479}
SPL {X  -159.990, Y  +446.037, Z    +0.000, E1   -23.324, E3 +480425.729}
SPL {X  -159.990, Y  +448.797, Z    +0.000, E1   -23.331, E3 +480439.260}
SPL {X  -159.990, Y  +451.747, Z    +0.000, E1   -23.333, E3 +480453.808}
SPL {X  -159.990, Y  +455.185, Z    +0.000, E1   -23.350, E3 +480470.668}
SPL {X  -159.990, Y  +458.265, Z    +0.000, E1   -23.328, E3 +480485.854}
SPL {X  -159.990, Y  +460.492, Z    +0.000, E1   -23.317, E3 +480496.853}
SPL {X  -159.990, Y  +462.929, Z    +0.000, E1   -23.331, E3 +480508.809}
SPL {X  -159.990, Y  +465.027, Z    +0.000, E1   -23.313, E3 +480519.162}
SPL {X  -159.990, Y  +466.881, Z    +0.000, E1   -23.322, E3 +480528.272}
SPL {X  -159.990, Y  +468.951, Z    +0.000, E1   -23.319, E3 +480538.464}
SPL {X  -159.990, Y  +471.818, Z    +0.000, E1   -23.351, E3 +480552.510}
SPL {X  -159.990, Y  +474.801, Z    +0.000, E1   -23.320, E3 +480567.286}
SPL {X  -159.990, Y  +476.830, Z    +0.000, E1   -23.323, E3 +480577.265}
SPL {X  -159.990, Y  +479.553, Z    +0.000, E1   -23.328, E3 +480590.667}
SPL {X  -159.990, Y  +482.950, Z    +0.000, E1   -23.350, E3 +480607.340}
SPL {X  -159.990, Y  +486.109, Z    +0.000, E1   -23.322, E3 +480622.955}
SPL {X  -159.990, Y  +488.481, Z    +0.000, E1   -23.319, E3 +480634.635}
SPL {X  -159.990, Y  +491.454, Z    +0.000, E1   -23.343, E3 +480649.215}
SPL {X  -159.990, Y  +494.937, Z    +0.000, E1   -23.343, E3 +480666.359}
SPL {X  -159.990, Y  +497.668, Z    +0.000, E1   -23.317, E3 +480679.852}
SPL {X  -159.990, Y  +499.995, Z    +0.000, E1   -23.324, E3 +480691.290}
SPL {X  -159.990, Y  +502.456, Z    +0.000, E1   -23.324, E3 +480703.405}
SPL {X  -159.990, Y  +504.508, Z    +0.000, E1   -23.311, E3 +480713.539}
SPL {X  -159.990, Y  +506.420, Z    +0.000, E1   -23.317, E3 +480722.932}
SPL {X  -159.990, Y  +508.862, Z    +0.000, E1   -23.328, E3 +480734.925}
SPL {X  -159.990, Y  +511.771, Z    +0.000, E1   -23.331, E3 +480749.246}
SPL {X  -159.990, Y  +514.016, Z    +0.000, E1   -23.308, E3 +480760.350}
SPL {X  -159.990, Y  +516.860, Z    +0.000, E1   -23.355, E3 +480774.236}
SPL {X  -159.990, Y  +520.719, Z    +0.000, E1   -23.363, E3 +480793.147}
SPL {X  -159.990, Y  +523.968, Z    +0.000, E1   -23.332, E3 +480809.231}
SPL {X  -159.990, Y  +526.466, Z    +0.000, E1   -23.320, E3 +480821.575}
SPL {X  -159.990, Y  +528.815, Z    +0.000, E1   -23.322, E3 +480833.134}
SPL {X  -159.990, Y  +531.246, Z    +0.000, E1   -23.325, E3 +480845.073}
SPL {X  -159.990, Y  +533.354, Z    +0.000, E1   -23.318, E3 +480855.458}
SPL {X  -159.990, Y  +534.931, Z    +0.000, E1   -23.312, E3 +480863.252}
SPL {X  -159.990, Y  +537.024, Z    +0.000, E1   -23.321, E3 +480873.551}
SPL {X  -159.990, Y  +539.129, Z    +0.000, E1   -23.310, E3 +480883.934}
SPL {X  -159.990, Y  +541.183, Z    +0.000, E1   -23.319, E3 +480894.031}
SPL {X  -159.990, Y  +544.314, Z    +0.000, E1   -23.352, E3 +480909.359}
SPL {X  -159.990, Y  +548.126, Z    +0.000, E1   -23.354, E3 +480928.114}
SPL {X  -159.990, Y  +551.344, Z    +0.000, E1   -23.327, E3 +480944.006}
SPL {X  -159.990, Y  +553.642, Z    +0.000, E1   -23.319, E3 +480955.325}
SPL {X  -159.990, Y  +556.481, Z    +0.000, E1   -23.354, E3 +480969.232}
SPL {X  -159.990, Y  +559.475, Z    +0.000, E1   -23.321, E3 +480984.038}
SPL {X  -159.990, Y  +561.830, Z    +0.000, E1   -23.325, E3 +480995.622}
SPL {X  -159.990, Y  +564.273, Z    +0.000, E1   -23.325, E3 +481007.646}
SPL {X  -159.990, Y  +566.342, Z    +0.000, E1   -23.314, E3 +481017.851}
SPL {X  -159.990, Y  +568.184, Z    +0.000, E1   -23.317, E3 +481026.912}
SPL {X  -159.990, Y  +570.560, Z    +0.000, E1   -23.333, E3 +481038.572}
SPL {X  -159.990, Y  +572.975, Z    +0.000, E1   -23.316, E3 +481050.491}
SPL {X  -159.990, Y  +575.097, Z    +0.000, E1   -23.325, E3 +481060.918}
SPL {X  -159.990, Y  +578.356, Z    +0.000, E1   -23.358, E3 +481076.890}
SPL {X  -159.990, Y  +582.292, Z    +0.000, E1   -23.360, E3 +481096.206}
SPL {X  -159.990, Y  +585.165, Z    +0.000, E1   -23.322, E3 +481110.449}
SPL {X  -159.990, Y  +587.388, Z    +0.000, E1   -23.328, E3 +481121.361}
SPL {X  -159.990, Y  +590.594, Z    +0.000, E1   -23.363, E3 +481137.053}
SPL {X  -159.990, Y  +594.301, Z    +0.000, E1   -23.358, E3 +481155.258}
SPL {X  -159.990, Y  +597.981, Z    +0.000, E1   -23.373, E3 +481173.306}
SPL {X  -159.990, Y  +600.935, Z    +0.000, E1   -23.343, E3 +481187.839}
SPL {X  -159.990, Y  +603.047, Z    +0.000, E1   -23.344, E3 +481198.224}
SPL {X  -159.990, Y  +605.187, Z    +0.000, E1   -23.344, E3 +481208.746}
SPL {X  -159.990, Y  +607.319, Z    +0.000, E1   -23.353, E3 +481219.209}
SPL {X  -159.990, Y  +610.569, Z    +0.000, E1   -23.372, E3 +481235.173}
SPL {X  -159.990, Y  +613.591, Z    +0.000, E1   -23.342, E3 +481250.102}
SPL {X  -159.990, Y  +615.604, Z    +0.000, E1   -23.330, E3 +481260.040}
SPL {X  -159.990, Y  +618.445, Z    +0.000, E1   -23.368, E3 +481273.953}
SPL {X  -159.990, Y  +621.517, Z    +0.000, E1   -23.337, E3 +481289.117}
SPL {X  -159.990, Y  +623.764, Z    +0.000, E1   -23.335, E3 +481300.168}
SPL {X  -159.990, Y  +625.941, Z    +0.000, E1   -23.337, E3 +481310.859}
SPL {X  -159.990, Y  +628.611, Z    +0.000, E1   -23.357, E3 +481323.938}
SPL {X  -159.990, Y  +631.169, Z    +0.000, E1   -23.338, E3 +481336.542}
SPL {X  -159.990, Y  +633.318, Z    +0.000, E1   -23.339, E3 +481347.131}
SPL {X  -159.990, Y  +635.650, Z    +0.000, E1   -23.339, E3 +481358.602}
SPL {X  -159.990, Y  +637.839, Z    +0.000, E1   -23.335, E3 +481369.413}
SPL {X  -159.990, Y  +640.072, Z    +0.000, E1   -23.325, E3 +481380.445}
SPL {X  -159.990, Y  +642.230, Z    +0.000, E1   -23.323, E3 +481391.126}
SPL {X  -159.990, Y  +645.287, Z    +0.000, E1   -23.340, E3 +481406.152}
SPL {X  -159.990, Y  +648.792, Z    +0.000, E1   -23.346, E3 +481423.411}
SPL {X  -159.990, Y  +652.623, Z    +0.000, E1   -23.348, E3 +481442.246}
SPL {X  -159.990, Y  +656.380, Z    +0.000, E1   -23.347, E3 +481460.740}
SPL {X  -159.990, Y  +659.180, Z    +0.000, E1   -23.314, E3 +481474.589}
SPL {X  -159.990, Y  +661.392, Z    +0.000, E1   -23.318, E3 +481485.482}
SPL {X  -159.990, Y  +663.662, Z    +0.000, E1   -23.322, E3 +481496.606}
SPL {X  -159.990, Y  +665.964, Z    +0.000, E1   -23.328, E3 +481507.897}
SPL {X  -159.990, Y  +668.989, Z    +0.000, E1   -23.359, E3 +481522.733}
SPL {X  -159.990, Y  +671.893, Z    +0.000, E1   -23.319, E3 +481537.113}
SPL {X  -159.974, Y  +673.789, Z    +0.000, E1   -23.323, E3 +481546.429}
SPL {X  -159.924, Y  +676.110, Z    +0.000, E1   -23.320, E3 +481557.913}
SPL {X  -159.801, Y  +679.265, Z    +0.000, E1   -23.327, E3 +481573.532}
SPL {X  -159.626, Y  +682.287, Z    +0.000, E1   -23.280, E3 +481588.630}
SPL {X  -159.462, Y  +684.486, Z    +0.000, E1   -23.258, E3 +481599.630}
SPL {X  -159.246, Y  +686.911, Z    +0.000, E1   -23.230, E3 +481611.791}
SPL {X  -159.019, Y  +689.098, Z    +0.000, E1   -23.200, E3 +481622.793}
SPL {X  -158.771, Y  +691.210, Z    +0.000, E1   -23.159, E3 +481633.469}
SPL {X  -158.553, Y  +692.896, Z    +0.000, E1   -23.130, E3 +481641.998}
ENDSPLINE

